				// Time out expected hanger is not arrived
				IF (me.SubStateMachine.udiTimeInState_ms > SIf.Par.udiTimeOutHRU_Hanger_ms) THEN	// Hanger Rotation Unit time out waiting
					pfbAlarmCtrl^.setAlarm(CIf.Info.intCtrlId,4,0,ADR(SIf.Alm),E_AlmState.RST,CIf.Job.eMe_ActivAlmClass);
					me.SubStateMachine.intStateNext := cSTA_SUB_ERROR;
				END_IF
		//--------------------------------------------------------------------------------------
			cSTA_SUB_WAIT_WITH_HANGER:
				IF (me.SubStateMachine.intState<>me.SubStateMachine.intStateLastCycle) THEN
					me.SubStateMachine.intStateLastCycle := me.SubStateMachine.intState;
				END_IF
				
				// State Change Condition
				// Check error if possible
				IF (me.SubStateMachine.udiTimeInState_ms >= SIf.Par.udiWaitForRotate_ms) THEN
					me.SubStateMachine.intStateNext := cSTA_SUB_ROTATE;
				END_IF
		//--------------------------------------------------------------------------------------
			cSTA_SUB_ROTATE:
				IF (me.SubStateMachine.intState<>me.SubStateMachine.intStateLastCycle) THEN
					me.SubStateMachine.intStateLastCycle := me.SubStateMachine.intState;
					SIf.Out.bolRotate.intern := NOT SIf.Out.bolRotate.intern;	// Rotate in other direction
				END_IF
				
				
				// State Change Condition
				// Check error if possible
				IF (me.SubStateMachine.udiTimeInState_ms >= SIf.Par.udiRotateTime_ms) THEN
					me.SubStateMachine.intStateNext := cSTA_SUB_EJECT;
				END_IF
		//--------------------------------------------------------------------------------------
			cSTA_SUB_EJECT:
				IF (me.SubStateMachine.intState<>me.SubStateMachine.intStateLastCycle) THEN
					me.SubStateMachine.intStateLastCycle := me.SubStateMachine.intState;
				END_IF
				
				SIf.Out.bolEject.intern := TRUE;	// Eject Cylinder Valve
				
				// Simulation
				IF (CIf.SwCfg.bolSimulation) THEN
					SIf.In.bolHangerDetected.intern := FALSE; // Hanger is leaving the HRU
				END_IF
				
				// State Change Condition
				// Check error if possible
				IF (me.SubStateMachine.udiTimeInState_ms > SIf.Par.udiEjectTime_ms) THEN
					IF (SIf.In.bolHangerDetected.intern) THEN
					// sensor Hanger detected always on
						pfbAlarmCtrl^.setAlarm(CIf.Info.intCtrlId,3,0,ADR(SIf.Alm),E_AlmState.RST,CIf.Job.eMe_ActivAlmClass);
						me.SubStateMachine.intStateNext := cSTA_SUB_ERROR;
					ELSE
						// Hanger ejected
						me.SubStateMachine.intStateNext := cSTA_SUB_RETRACT;
					END_IF
				END_IF
		//--------------------------------------------------------------------------------------
			cSTA_SUB_RETRACT:
				IF (me.SubStateMachine.intState<>me.SubStateMachine.intStateLastCycle) THEN
					me.SubStateMachine.intStateLastCycle := me.SubStateMachine.intState;
				END_IF
				
				SIf.Out.bolEject.intern := FALSE;	// Eject Cylinder Valve

				// State Change Condition
				// Check error if possible
				IF (me.SubStateMachine.udiTimeInState_ms >= SIf.Par.udiRetractTime_ms) THEN
					me.SubStateMachine.intStateNext := cSTA_SUB_DONE;
				END_IF
		//--------------------------------------------------------------------------------------
			cSTA_SUB_DONE:
				//CIf.Job.intACmd:=cSTA_DONE; 	// Not necessary
				;								// do nothing, just for state change
		//--------------------------------------------------------------------------------------
			cSTA_SUB_ERROR:
				IF (me.SubStateMachine.intState<>me.SubStateMachine.intStateLastCycle) THEN
					me.SubStateMachine.intStateLastCycle := me.SubStateMachine.intState;
				END_IF
				
				SIf.Out.bolEject.intern := FALSE;	// Eject Cylinder Valve
				
				// State Change Condition
				// No change, going over an other main state
		//--------------------------------------------------------------------------------------
		END_CASE
		
		// Do in every cycle
		CIf.Job.strSubState := THIS^.getCmdState(intCmdState:=me.SubStateMachine.intState,bolState:=TRUE);
		IF (me.SubStateMachine.intState<>me.SubStateMachine.intStateNext) THEN
			me.SubStateMachine.intState := me.SubStateMachine.intStateNext;  // set next state for next cycle
			me.SubStateMachine.udiTimeInState_ms := 0; // reset timer
			// log state change -> open point
		ELSE
			// increment time in state	
			me.SubStateMachine.udiTimeInState_ms := me.SubStateMachine.udiTimeInState_ms + me.FUBInfo.udiSample_ms;
		END_IF
		
				
		// State Change Condition	
		IF me.SubStateMachine.intState = cSTA_SUB_ERROR THEN
			me.StateMachine.intStateNext :=  cSTA_ERROR;
		ELSIF(me.SubStateMachine.intState = cSTA_SUB_DONE) THEN
			me.StateMachine.intStateNext := cSTA_RUN;
		ELSIF((me.SubStateMachine.intState = cSTA_SUB_WAIT_FOR_JOB) AND(me.intCmd=cCMD_STOP)) THEN
			me.StateMachine.intStateNext := cSTA_STOPBusy;
		//ELSIF((me.SubStateMachine.intState = cSTA_SUB_WAIT_FOR_JOB) AND(me.intCmd=cCMD_OFF)) THEN // Done by BaseCtrl.Always
		//	me.StateMachine.intStateNext := cSTA_OFFBusy;
		END_IF
	END_IF


//--------------------------------------------------------------------------------------
// Exit action
	IF (me.StateMachine.intState<>me.StateMachine.intStateNext) THEN
		;
	END_IF
END_METHOD

METHOD PROTECTED sta_STOP : BOOL
// state implemetation
//--------------------------------------------------------------------------------------
// Entry action
	IF (me.StateMachine.intState<>me.StateMachine.intStateLastCycle) THEN
		me.StateMachine.intStateLastCycle := me.StateMachine.intState;
		
	END_IF


//--------------------------------------------------------------------------------------
// Cyclic action
	IF (me.StateMachine.intState=me.StateMachine.intStateLastCycle) THEN
		
		;
		
		
		// State Change Condition
		IF (me.intCmd=cCMD_OFF) THEN
			// sensor retract always on cylinder
			me.StateMachine.intStateNext :=  cSTA_OFFBusy;
		ELSIF (me.intCmd=cCMD_EJECT) THEN 
			me.StateMachine.intStateNext := cSTA_EJECTBusy;
		ELSIF(me.intCmd=cCMD_RETRACT) THEN
			me.StateMachine.intStateNext := cSTA_RETRACTBusy;
		ELSIF(me.intCmd=cCMD_ROTATE) THEN
			me.StateMachine.intStateNext := cSTA_ROTATEBusy;
		ELSIF (me.intCmd=cCMD_RUN) THEN
			me.StateMachine.intStateNext := cSTA_RUNBusy;
		END_IF
	END_IF




//--------------------------------------------------------------------------------------
// Exit action
	IF (me.StateMachine.intState<>me.StateMachine.intStateNext) THEN
		;
	END_IF
END_METHOD

METHOD PROTECTED sta_STOPBusy : BOOL
// state implemetation
//--------------------------------------------------------------------------------------
// Entry action
	IF (me.StateMachine.intState<>me.StateMachine.intStateLastCycle) THEN
		me.StateMachine.intStateLastCycle := me.StateMachine.intState;
		
	END_IF


//--------------------------------------------------------------------------------------
// Cyclic action
	IF (me.StateMachine.intState=me.StateMachine.intStateLastCycle) THEN
		
		// switch off?
		// SIf.Out.bolEject.intern := FALSE;	// Eject Cylinder Valve
		
		// State Change Condition
		IF (FALSE) THEN
			;
		ELSIF (TRUE) THEN
			me.StateMachine.intStateNext := cSTA_STOP;
		END_IF
	END_IF




//--------------------------------------------------------------------------------------
// Exit action
	IF (me.StateMachine.intState<>me.StateMachine.intStateNext) THEN
		;
	END_IF
END_METHOD

METHOD PROTECTED StateMachine : BOOL
SUPER^.StateMachine();

// main statemachine of base controller
CASE me.StateMachine.intState OF
	cSTA_ROTATEBusy: 
        THIS^.sta_ROTATEBusy();
    cSTA_ROTATE: 
        THIS^.sta_ROTATE();
	cSTA_RETRACTBusy: 
        THIS^.sta_RETRACTBusy();
    cSTA_RETRACT: 
        THIS^.sta_RETRACT();
    cSTA_EJECTBusy:				// Eject 
        THIS^.sta_EJECTBusy();
    cSTA_EJECT: 
        THIS^.sta_EJECT();
	cSTA_RUNBusy: 
        THIS^.sta_RUNBusy();	// Auto (Wait - Rotate - Eject - Retract)
    cSTA_RUN: 
        THIS^.sta_RUN();
	cSTA_STOPBusy: 				// Rotate rests in his Position, Ejector in Retract Position
        THIS^.sta_STOPBusy();
    cSTA_STOP: 
        THIS^.sta_STOP();
		
END_CASE;
END_METHOD

END_FUNCTION_BLOCK

// POUs/Controller/Lvl0/JUN (Junction)/FB_JUN
FUNCTION_BLOCK FB_JUN EXTENDS FB_CtrlBase
VAR_INPUT
	In_bolPassed: BOOL;
END_VAR
VAR_OUTPUT
	Out_bolOpen: BOOL;
END_VAR
VAR
	/// Specific interface struct for public access
	SIf: T_Ctrl_SIf_JUN;
	/// Function specific variables
	bolfpRelease: BOOL;
	/// Job for checking the sensor
	bolCheckPass: BOOL;
	/// standard Loop variable
	uinI: UINT;
	/// Loop Variable for Hashtable
	intLoopHashtable: INT;
	/// Index to next job in Hashtable
	intNextHastableIdx: INT;
	/// Index to next job in Hashtable
	intActHastableIdx: INT;
	/// Calculated position to open junction
	dinNextOpenPosition_um: DINT;
	/// Calculated position to close junction
	dinNextClosePosition_um: DINT;
	///Last new position value from parent
	dinTransportPositionOld_um: DINT;
	///Position correction in faster Task cycletime
	dinPositionCorrection_um: DINT;
	///Position of the tag
	dinTagPosition_um: DINT;
	///Difference from actual Tag Position to junction
	dinPositionDifference_um: DINT;
	/// Rising edge of passed sensor
	bolFpPassed: BOOL;
	/// Array to check every hanger passed the sensor
	aCheckPassingTime: ARRAY[0..9] OF T_JUN_OutfeedCheck;
	/// Size of Array Check Passing
	intSizeCheckPassing: INT;
	/// Index for the check passing array
	intIndexCheckPassing: INT;
	/// Temporary Value
	udiValue: UDINT;
	/// Temporary Value
	uinValue: UINT;
END_VAR
VAR CONSTANT
	///sub States for RELEASE Function
	cSTA_SUB_INITIALIZED: INT := 500;
	cSTA_SUB_WAIT_FOR_JOB: INT := 501;
	cSTA_SUB_OPEN: INT := 502;
	cSTA_SUB_CLOSE: INT := 506;
	cSTA_SUB_ERROR: INT := 598;
	cSTA_SUB_FINISHED: INT := 600;
END_VAR

(*__________________________________________________________________________________________________
¦	
¦	Vistaprint Schweiz GmbH
¦	CH - 8401 Winterthur
¦
¦	www.vistaprint.ch - info@vistaprint.ch
¦___________________________________________________________________________________________________

Function desription:
Junction to release hanges out of the transport belt 


History:
Version		Date			Author		Comment
---------------------------------------------------------------------------------------------------
0.00.1		22.08.2013		AVME/PRE	Start history
0.00.2		19.09.2013		AVME/PRE	Implement new Base Concept
0.00.3		02.10.2013		VP/MK,RE	Fixed multiplication issues (cast INT to REAL before division)
0.00.4		10.12.2013		AVME/MRU	Reset aCheckPassing time at exit of sta_RUN
0.00.5		03.02.2014		AVME/MRU	Changed 'timeout passed sensor does not detect the hanger' to INFO

___________________________________________________________________________________________________*)


IF (me.bolActivate) THEN // cyclic call enabled
	IF (CIf.Info.bolInitDone=FALSE) THEN // first cycle -> init
		CtrlInit();
		CIf.Info.bolInitDone := TRUE;
	ELSE
		CycleStartDuty();
	
		Always();
		
		StateMachine();
		
		CycleEndDuty();
	END_IF
END_IF;

METHOD PROTECTED Always : BOOL
IF (me.bolChangeBackToAUTO=TRUE) THEN // switch mode to automatic switch off controller
	//me.StateMachine.intStateNext := cSTA_OFFBusy;
	me.bolChangeBackToAUTO := FALSE; // for cylinder no change to off when switch to automatic!!
END_IF

SUPER^.Always();

// ----------------------------------------------------------------------------------
// cyclic actions outside of statemachine
IF (me.StateMachine.intState<>cSTA_SINGLE_ANSWER) THEN
	SIf.Cur.bolPassed := SIf.In.bolPassed.intern;
	SIf.Cur.bolOpen := SIf.Out.bolOpen.intern;

	; // always error supervision
	
END_IF

// Always change actions in Base Library
// ----------------------------------------------------------------------------------
// overrule error always from base -> no EOFF State!! in EOFF go to OFF
IF (me.StateMachine.intStateNext = cSTA_EOFFBusy) THEN
	IF (me.StateMachine.intState=cSTA_OFF) THEN
		me.StateMachine.intStateNext := cSTA_OFF;
	ELSE // stay in OFF
		me.StateMachine.intStateNext := cSTA_OFFBusy;
	END_IF
END_IF
END_METHOD

METHOD FB_init : BOOL
VAR_INPUT
	///if TRUE, the retain variables are initialized (warm start / cold start)
	bInitRetains: BOOL;
	///if TRUE, the instance afterwards gets moved into the copy code (online change)
	bInCopyCode: BOOL;
END_VAR
VAR
	ii: UINT;
END_VAR
//------------------------------------------------------------------------------------------------------------------------
// to manually change in new FUB implementation!!!
// define valid commands for this controller
FOR ii:= 0 TO (SIZEOF(CIf.Job.aCmdList)/SIZEOF(CIf.Job.aCmdList[0])-1) BY 1 DO
	IF (CIf.Job.aCmdList[ii].intCmd=cCMD_INITIALIZED) THEN
		// found first empty array element
		EXIT;
	END_IF
END_FOR
CIf.Job.aCmdList[ii].intCmd := cCMD_STOP;
CIf.Job.aCmdList[ii].strName := 'Stop'; 
CIf.Job.aCmdList[ii].bolAvailable := TRUE;
ii := ii +1;
CIf.Job.aCmdList[ii].intCmd := JUN_CmdState.cCMD_RELEASE_ALL;
CIf.Job.aCmdList[ii].strName := 'Release All';
CIf.Job.aCmdList[ii].bolAvailable := TRUE;
ii := ii +1;
CIf.Job.aCmdList[ii].intCmd := JUN_CmdState.cCMD_RELEASE; // for test simulation single answer
CIf.Job.aCmdList[ii].strName := 'Release';
CIf.Job.aCmdList[ii].bolAvailable := TRUE;
ii := ii +1;
CIf.Job.aCmdList[ii].intCmd := cCMD_RUN;
CIf.Job.aCmdList[ii].strName := 'Run'; 
CIf.Job.aCmdList[ii].bolAvailable := TRUE;
ii := ii +1;
CIf.Job.aCmdList[ii].intCmd := cCMD_STOP;
CIf.Job.aCmdList[ii].strName := 'Stop'; 
CIf.Job.aCmdList[ii].bolAvailable := TRUE;
ii := ii +1;

// set name of class/typ
CIf.Info.strType := 'FB_JUN'; 

// set alarm class
SIf.Alm[1].eAlmClass := E_AlmClass.INFO;
SIf.Alm[1].strText := 'timeout passed sensor does not detect the hanger'; 
SIf.Alm[2].eAlmClass := E_AlmClass.INFO;
SIf.Alm[2].strText := 'RUN not possible, no Hashtable';
SIf.Alm[3].eAlmClass := E_AlmClass.INFO;
SIf.Alm[3].strText := 'Open not possible, destination is full';
SIf.Alm[4].eAlmClass := E_AlmClass.TSTOP;
SIf.Alm[4].strText := 'interlock open - movement stopped';


//*******************************************************************************
// initial values
//*******************************************************************************

// software configuration
CIf.SwCfg.bolExist := TRUE;
CIf.SwCfg.bolSimulation := FALSE;

// parmeter
SIf.Par.udiOpenTime_ms := 20;
SIf.Par.udiCloseTime_ms := 10;
SIf.Par.udiPassTime_ms := 6000;

SIf.Par.udiSimPassTime_ms := SIf.Par.udiPassTime_ms/2;

SIf.Par.dinPosition_um := 10000000;
SIf.Par.dinOpenWay_um := 200000;

//*******************************************************************************
// initial values childes
//*******************************************************************************
END_METHOD

METHOD PROTECTED getCmdState : STRING
VAR_INPUT
	intCmdState: INT;
	bolState: BOOL;
END_VAR
getCmdState := SUPER^.getCmdState(intCmdState:=intCmdState,bolState:=bolState); // get global/base defined cmds/states
IF (getCmdState='') THEN // global not defined get local
	// get string cmd/state string information in runtime
	IF (bolState=FALSE) THEN
		// cmd's
		CASE intCmdState OF
			JUN_CmdState.cCMD_RELEASE_ALL: 
				getCmdState := 'cCMD_RELEASE_ALL';
			JUN_CmdState.cCMD_RELEASE: 
				getCmdState := 'cCMD_RELEASE';
		END_CASE;
	ELSE
	
	// cmd's
		CASE intCmdState OF
			cSTA_RUNBusy: 
				THIS^.sta_RUNBusy();
			cSTA_RUN: 
				THIS^.sta_RUN();
			cSTA_STOPBusy: 
				THIS^.sta_STOPBusy();
			cSTA_STOP: 
				THIS^.sta_STOP();
			JUN_CmdState.cSTA_RELEASE_ALLBusy: 
				THIS^.sta_RELEASE_ALLBusy();
			JUN_CmdState.cSTA_RELEASE_ALL: 
				THIS^.sta_RELEASE_ALL();
			JUN_CmdState.cSTA_RELEASEBusy: 
				THIS^.sta_RELEASEBusy();
			JUN_CmdState.cSTA_RELEASE: 
				THIS^.sta_RELEASE();
				
			// SUB States
			cSTA_SUB_INITIALIZED:
				getCmdState := 'cSTA_SUB_INITIALIZED';
			cSTA_SUB_WAIT_FOR_JOB:
				getCmdState := 'cSTA_SUB_WAIT_FOR_JOB';
			cSTA_SUB_OPEN:
				getCmdState := 'cSTA_SUB_OPEN';
			cSTA_SUB_CLOSE:
				getCmdState := 'cSTA_SUB_CLOSE';
			cSTA_SUB_ERROR:
				getCmdState := 'cSTA_SUB_ERROR';
			cSTA_SUB_FINISHED:
				getCmdState := 'cSTA_SUB_FINISHED';
		END_CASE;
	END_IF
END_IF
END_METHOD

METHOD getCtrlSIf : POINTER TO T_Ctrl_SIf_JUN
getCtrlSIf := ADR(SIf);
END_METHOD

METHOD PROTECTED IoInBridge : BOOL
// digitale and analoge inputs read from hardware or forcing

SIf.In.bolPassed.map := THIS^.In_bolPassed;

IF (CIf.SwCfg.bolSimulation = FALSE) THEN
	getInBol(CIf.Job.bolIoForce,ADR(SIf.In.bolPassed));
	//ctrl.In.bol_PosSwitchBasicDefTyp.intern := getInBol(ctrl.ifc.Job.bol_Force ,ADR(ctrl.In.bol_PosSwitchBasicDefTyp);
ELSE
	//simulation of global IO
END_IF
END_METHOD

METHOD PROTECTED IoOutBridge : BOOL
// digitale and analoge inputs read from hardware or forcing
IF (CIf.SwCfg.bolSimulation = FALSE) THEN
	setOutBol(CIf.Job.bolIoForce ,ADR(SIf.Out.bolOpen));
	
	// check interlocks to prevent damages
	IF (CIf.Job.bolIlkOverwrite=FALSE) THEN
		IF (SIf.Ilk.bolOpen=TRUE) THEN
			// switch off?
			IF (SIf.Out.bolOpen.map = TRUE) THEN
				// Set alarm: SIf.Alm[4].strText := 'interlock open - movement stopped';
				pfbAlarmCtrl^.setAlarm(CIf.Info.intCtrlId,4,0,ADR(SIf.Alm),E_AlmState.RST,CIf.Job.eMe_ActivAlmClass);
			END_IF
			SIf.Out.bolOpen.map := FALSE;
		END_IF	
	END_IF
	THIS^.Out_bolOpen := SIf.Out.bolOpen.map;
END_IF
END_METHOD

METHOD PROTECTED sta_ERROR : BOOL
// state implemetation
//--------------------------------------------------------------------------------------
// Entry action
	IF (me.StateMachine.intState<>me.StateMachine.intStateLastCycle) THEN
		me.StateMachine.intStateHistory := me.StateMachine.intStateLastCycle; // -> possibillity to go back to state before error
		me.StateMachine.intStateLastCycle := me.StateMachine.intState;
		
	END_IF


//--------------------------------------------------------------------------------------
// Cyclic action
	IF (me.StateMachine.intState=me.StateMachine.intStateLastCycle) THEN
		
		SIf.Out.bolOpen.intern := 0;
		
		
		// State Change Condition
		IF (CIf.Job.bolAlmReset = TRUE) THEN
			me.StateMachine.intStateNext := cSTA_ERRORQuit;
		END_IF
	END_IF




//--------------------------------------------------------------------------------------
// Exit action
	IF (me.StateMachine.intState<>me.StateMachine.intStateNext) THEN
		;
	END_IF
END_METHOD

METHOD PROTECTED sta_ERRORQuit : BOOL
// state implemetation
//--------------------------------------------------------------------------------------
// Entry action
	IF (me.StateMachine.intState<>me.StateMachine.intStateLastCycle) THEN
		me.StateMachine.intStateLastCycle := me.StateMachine.intState;
			FOR uinI := 0 TO (SIZEOF(aCheckPassingTime)/(SIZEOF(aCheckPassingTime[0]))-1) DO
				aCheckPassingTime[uinI].udiTime_ms := 0;
				aCheckPassingTime[uinI].intHTIndex := 0;
			END_FOR
	END_IF


//--------------------------------------------------------------------------------------
// Cyclic action
	IF (me.StateMachine.intState=me.StateMachine.intStateLastCycle) THEN
		
		;
		// evtl. wait time if reset of device is necessary and then decide to go to states or ERROR state
		IF (CIf.Job.bolAlmReset = TRUE) THEN
			CIf.Job.eMe_ActivAlmClass := E_AlmClass.NONE; // reset feedback channel for parent
			CIf.Job.bolAlmReset := FALSE;
		END_IF
		
		// State Change Condition
		IF (CIf.Job.bolAlmReset = FALSE) THEN
			IF (me.StateMachine.intStateHistory<=cSTA_PON) THEN
				me.StateMachine.intStateNext := cSTA_PONBusy;
			ELSIF(me.intCmd=cCMD_OFF) THEN
				me.StateMachine.intStateNext := cSTA_OFFBusy;
			ELSIF(me.intCmd=cCMD_RUN) OR (me.StateMachine.intStateHistory=cSTA_RUN) THEN
				me.StateMachine.intStateNext := cSTA_RUNBusy;
			ELSIF(me.intCmd=cCMD_STOP) THEN
				me.StateMachine.intStateNext := cSTA_STOPBusy;
			ELSIF(me.intCmd=JUN_CmdState.cCMD_RELEASE_ALL) THEN
				me.StateMachine.intStateNext := JUN_CmdState.cSTA_RELEASE_ALLBusy;
			ELSIF(me.intCmd=JUN_CmdState.cCMD_RELEASE) THEN
				me.StateMachine.intStateNext := JUN_CmdState.cSTA_RELEASEBusy;
			END_IF
		END_IF
	END_IF




//--------------------------------------------------------------------------------------
// Exit action
	IF (me.StateMachine.intState<>me.StateMachine.intStateNext) THEN
		;
	END_IF
END_METHOD

METHOD PROTECTED sta_OFF : BOOL
// state implemetation
//--------------------------------------------------------------------------------------
// Entry action
	IF (me.StateMachine.intState<>me.StateMachine.intStateLastCycle) THEN
		me.StateMachine.intStateLastCycle := me.StateMachine.intState;
		
	END_IF


//--------------------------------------------------------------------------------------
// Cyclic action
	IF (me.StateMachine.intState=me.StateMachine.intStateLastCycle) THEN
		
		;
		
		
		// State Change Condition
		IF (me.Alarm.eActivAlmClass<>E_AlmClass.EOFF) AND (me.Alarm.eActivAlmClass<>E_AlmClass.OFF) THEN
			IF (me.intCmd=cCMD_STOP) THEN
				// sensor retract always on cylinder
				me.StateMachine.intStateNext :=  cSTA_STOPBusy;
			ELSIF (me.intCmd=JUN_CmdState.cCMD_RELEASE) THEN 
				me.StateMachine.intStateNext := JUN_CmdState.cSTA_RELEASEBusy;
			ELSIF(me.intCmd=JUN_CmdState.cCMD_RELEASE_ALL) THEN
				me.StateMachine.intStateNext := JUN_CmdState.cSTA_RELEASE_ALLBusy;
			ELSIF(me.intCmd=cCMD_RUN) THEN
				me.StateMachine.intStateNext := cSTA_RUNBusy;
			END_IF
		END_IF
	END_IF




//--------------------------------------------------------------------------------------
// Exit action
	IF (me.StateMachine.intState<>me.StateMachine.intStateNext) THEN
		;
	END_IF
END_METHOD

METHOD PROTECTED sta_OFFBusy : BOOL
// state implemetation
//--------------------------------------------------------------------------------------
// Entry action
	IF (me.StateMachine.intState<>me.StateMachine.intStateLastCycle) THEN
		me.StateMachine.intStateLastCycle := me.StateMachine.intState;
		
	END_IF


//--------------------------------------------------------------------------------------
// Cyclic action
	IF (me.StateMachine.intState=me.StateMachine.intStateLastCycle) THEN
		
		// switch VALVE off
		SIf.Out.bolOpen.intern := FALSE;
		
		
		
		// State Change Condition
		IF (FALSE) THEN
			;
		ELSIF (TRUE) THEN
			me.StateMachine.intStateNext := cSTA_OFF;
		END_IF
	END_IF




//--------------------------------------------------------------------------------------
// Exit action
	IF (me.StateMachine.intState<>me.StateMachine.intStateNext) THEN
		;
	END_IF
END_METHOD

METHOD PROTECTED sta_PON : BOOL
// state implemetation
//--------------------------------------------------------------------------------------
// Entry action
	IF (me.StateMachine.intState<>me.StateMachine.intStateLastCycle) THEN
		me.StateMachine.intStateLastCycle := me.StateMachine.intState;
		
	END_IF


//--------------------------------------------------------------------------------------
// Cyclic action
	IF (me.StateMachine.intState=me.StateMachine.intStateLastCycle) THEN
		
		;
		
		
		// State Change Condition
		IF(me.intCmd=cCMD_OFF) THEN
			me.StateMachine.intStateNext := cSTA_OFFBusy;
		ELSIF(me.intCmd=cCMD_RUN) THEN
			me.StateMachine.intStateNext := cSTA_OFFBusy;
		ELSIF(me.intCmd=cCMD_STOP) THEN
			me.StateMachine.intStateNext := cSTA_STOPBusy;
		ELSIF(me.intCmd=JUN_CmdState.cCMD_RELEASE) THEN
			me.StateMachine.intStateNext := JUN_CmdState.cSTA_RELEASEBusy;
		ELSIF (me.intCmd=JUN_CmdState.cCMD_RELEASE_ALL) THEN
			me.StateMachine.intStateNext := JUN_CmdState.cSTA_RELEASE_ALLBusy;
		END_IF
	END_IF




//--------------------------------------------------------------------------------------
// Exit action
	IF (me.StateMachine.intState<>me.StateMachine.intStateNext) THEN
		;
	END_IF
END_METHOD

METHOD PROTECTED sta_RELEASE : BOOL
// state implemetation
//--------------------------------------------------------------------------------------
// Entry action
	IF (me.StateMachine.intState<>me.StateMachine.intStateLastCycle) THEN
		me.StateMachine.intStateLastCycle := me.StateMachine.intState;
		
	END_IF


//--------------------------------------------------------------------------------------
// Cyclic action
	IF (me.StateMachine.intState=me.StateMachine.intStateLastCycle) THEN
		// Check the CMD change for next release
		IF (me.intCmd<>JUN_CmdState.cCMD_RELEASE) THEN
			bolfpRelease := FALSE;		// Only start once the release if cmd is still the same
		END_IF
	
	
		// Simulation
		
		// State Change Condition
		IF(me.intCmd=cCMD_STOP) THEN
			me.StateMachine.intStateNext := cSTA_STOPBusy;
		ELSIF(me.intCmd=JUN_CmdState.cCMD_RELEASE_ALL) THEN
			me.StateMachine.intStateNext := JUN_CmdState.cSTA_RELEASE_ALLBusy;
		ELSIF((me.intCmd=JUN_CmdState.cCMD_RELEASE) AND (bolfpRelease = FALSE)) THEN
			me.StateMachine.intStateNext := JUN_CmdState.cSTA_RELEASEBusy;			
		ELSIF(me.intCmd=cCMD_RUN) THEN
			me.StateMachine.intStateNext := cSTA_STOPBusy;			
		END_IF
	END_IF




//--------------------------------------------------------------------------------------
// Exit action
	IF (me.StateMachine.intState<>me.StateMachine.intStateNext) THEN
		bolfpRelease := FALSE;		// Only start once the release if cmd is still the same
	END_IF
END_METHOD

METHOD PROTECTED sta_RELEASE_ALL : BOOL
// state implemetation
//--------------------------------------------------------------------------------------
// Entry action
	IF (me.StateMachine.intState<>me.StateMachine.intStateLastCycle) THEN
		me.StateMachine.intStateLastCycle := me.StateMachine.intState;
		
		fbSimulationTimer.IN := FALSE;
		fbSimulationTimer.PT := UDINT_TO_TIME(SIf.Par.udiSimPassTime_ms);
		fbSimulationTimer(); // set time/reset timer
		fbSimulationTimer.IN := TRUE; // start timer

	END_IF


//--------------------------------------------------------------------------------------
// Cyclic action
	IF (me.StateMachine.intState=me.StateMachine.intStateLastCycle) THEN

		// Simulation
		IF (CIf.SwCfg.bolSimulation) THEN
			fbSimulationTimer(); // simulation time
			IF (fbSimulationTimer.Q) THEN
				fbSimulationTimer.IN := FALSE;
				IF SIf.In.bolPassed.intern = FALSE THEN
					SIf.In.bolPassed.intern := TRUE;
				ELSE
					SIf.In.bolPassed.intern := FALSE;
				END_IF
			ELSE
				fbSimulationTimer.IN := TRUE; // start timer
			END_IF
		END_IF

		
		// State Change Condition
		IF(me.intCmd=cCMD_STOP) THEN
			me.StateMachine.intStateNext := cSTA_STOPBusy;
		ELSIF(me.intCmd=JUN_CmdState.cCMD_RELEASE) THEN
			me.StateMachine.intStateNext := JUN_CmdState.cSTA_RELEASEBusy;
		ELSIF(me.intCmd=cCMD_RUN) THEN
			me.StateMachine.intStateNext := cSTA_STOPBusy;
		END_IF
	END_IF




//--------------------------------------------------------------------------------------
// Exit action
	IF (me.StateMachine.intState<>me.StateMachine.intStateNext) THEN
		;
	END_IF
END_METHOD

METHOD PROTECTED sta_RELEASE_ALLBusy : BOOL
// state implemetation
//--------------------------------------------------------------------------------------
// Entry action
	IF (me.StateMachine.intState<>me.StateMachine.intStateLastCycle) THEN
		me.StateMachine.intStateLastCycle := me.StateMachine.intState;
		
		SIf.Out.bolOpen.intern := TRUE;
	END_IF


//--------------------------------------------------------------------------------------
// Cyclic action
	IF (me.StateMachine.intState=me.StateMachine.intStateLastCycle) THEN

		// Simulation

		
		// State Change Condition
		IF (me.StateMachine.udiTimeInState_ms > SIf.Par.udiOpenTime_ms) THEN
			me.StateMachine.intStateNext := JUN_CmdState.cSTA_RELEASE_ALL;
		ELSIF(me.intCmd=cCMD_STOP) THEN
			me.StateMachine.intStateNext := cSTA_STOPBusy;
		ELSIF(me.intCmd=JUN_CmdState.cCMD_RELEASE) THEN
			me.StateMachine.intStateNext := JUN_CmdState.cSTA_RELEASEBusy;
		ELSIF(me.intCmd=cCMD_RUN) THEN
			me.StateMachine.intStateNext := cSTA_STOPBusy;
		END_IF
	END_IF




//--------------------------------------------------------------------------------------
// Exit action
	IF (me.StateMachine.intState<>me.StateMachine.intStateNext) THEN
		;
	END_IF
END_METHOD

METHOD PROTECTED sta_RELEASEBusy : BOOL
// state implemetation
//--------------------------------------------------------------------------------------
// Entry action
	IF (me.StateMachine.intState<>me.StateMachine.intStateLastCycle) THEN
		me.StateMachine.intStateLastCycle := me.StateMachine.intState;
					
		me.SubStateMachine.intState := cSTA_SUB_INITIALIZED; // init sub state machine
		me.SubStateMachine.intStateNext := cSTA_SUB_INITIALIZED; // init sub state machine
		bolfpRelease := TRUE;		// Only start once the release if cmd is still the same
	END_IF


//--------------------------------------------------------------------------------------
// Cyclic action
	IF (me.StateMachine.intState=me.StateMachine.intStateLastCycle) THEN
	

		//--------------------------------------------------------------------------------------
		// sub state machine for sequence
		CASE me.SubStateMachine.intState OF
			//--------------------------------------------------------------------------------------
			cSTA_SUB_INITIALIZED:
					// State Change Condition
					// Simulation
					IF (CIf.SwCfg.bolSimulation) THEN
							SIf.In.bolPassed.intern := FALSE;
					END_IF

					// only release one tray if no jam is at the stopper
					IF (SIf.In.bolPassed.intern = FALSE) THEN
						me.SubStateMachine.intStateNext := cSTA_SUB_OPEN;
						// Start Timer
						fbSimulationTimer.IN := FALSE;
						fbSimulationTimer.PT := UDINT_TO_TIME(SIf.Par.udiSimPassTime_ms);
						fbSimulationTimer(); // set time/reset timer
						fbSimulationTimer.IN := TRUE; // start timer
	
					ELSE
						// SIf.Alm[3].strText := 'Open not possible, destination is full';
						pfbAlarmCtrl^.setAlarm(CIf.Info.intCtrlId,3,0,ADR(SIf.Alm),E_AlmState.RST,CIf.Job.eMe_ActivAlmClass);	
					END_IF
					
			//--------------------------------------------------------------------------------------
			cSTA_SUB_OPEN:
					SIf.Out.bolOpen.intern := TRUE;
					
					// Simulation
					IF (CIf.SwCfg.bolSimulation) THEN
						fbSimulationTimer(); // simulation time
						IF (fbSimulationTimer.Q) THEN
							SIf.In.bolPassed.intern := TRUE;						
						END_IF
					END_IF
					
					
				// State Change Condition
					// Check error if tray never reach the output
					IF (me.SubStateMachine.udiTimeInState_ms>SIf.Par.udiPassTime_ms) THEN
						// Set Alarm: SIf.Alm[1].strText := 'timeout passed sensor does not detect the hanger'; 
						pfbAlarmCtrl^.setAlarm(CIf.Info.intCtrlId,1,0,ADR(SIf.Alm),E_AlmState.RST,CIf.Job.eMe_ActivAlmClass);
						me.SubStateMachine.intStateNext := cSTA_ERROR;
					// Check if tray allready passed
					ELSIF (SIf.In.bolPassed.intern = TRUE) THEN
						me.SubStateMachine.intStateNext := cSTA_SUB_CLOSE;
					END_IF

					
			//--------------------------------------------------------------------------------------
			cSTA_SUB_CLOSE:
					SIf.Out.bolOpen.intern := FALSE;
					
					// Simulation
					
					
					// State Change Condition
					// Check error if retracted position not reached
					IF (me.SubStateMachine.udiTimeInState_ms > SIf.Par.udiCloseTime_ms) THEN
						me.SubStateMachine.intStateNext := cSTA_SUB_FINISHED;
						// Simulation
						IF (CIf.SwCfg.bolSimulation) THEN
								SIf.In.bolPassed.intern := FALSE;
						END_IF
					END_IF
				
			//--------------------------------------------------------------------------------------
			cSTA_SUB_ERROR:
					SIf.Out.bolOpen.intern := FALSE;
					
					// State Change Condition
					// No change, going over an other main state
					
			//--------------------------------------------------------------------------------------
			cSTA_SUB_FINISHED:
					;
					
		END_CASE
		
		// State Change Condition
		// Check error if retracted position not reached
		IF me.SubStateMachine.intState = cSTA_SUB_ERROR THEN
			me.StateMachine.intStateNext :=  cSTA_ERROR;
		ELSIF (me.SubStateMachine.intState = cSTA_SUB_FINISHED) THEN
			me.StateMachine.intStateNext := JUN_CmdState.cSTA_RELEASE;
		ELSIF(me.intCmd=cCMD_STOP) THEN
			me.StateMachine.intStateNext := cSTA_STOPBusy;
		ELSIF(me.intCmd=JUN_CmdState.cCMD_RELEASE_ALL) THEN
			me.StateMachine.intStateNext := JUN_CmdState.cSTA_RELEASE_ALLBusy;
		ELSIF(me.intCmd=cCMD_RUN) THEN
			me.StateMachine.intStateNext := cSTA_STOPBusy;			
		END_IF
	END_IF




//--------------------------------------------------------------------------------------
// Exit action
	IF (me.StateMachine.intState<>me.StateMachine.intStateNext) THEN
		;
	END_IF
END_METHOD

METHOD PROTECTED sta_RUN : BOOL
// state implemetation
//--------------------------------------------------------------------------------------
// Entry action
	IF (me.StateMachine.intState<>me.StateMachine.intStateLastCycle) THEN
		me.StateMachine.intStateLastCycle := me.StateMachine.intState;
			
		me.SubStateMachine.intState := cSTA_SUB_WAIT_FOR_JOB; // init sub state machine
		me.SubStateMachine.intStateNext := cSTA_SUB_WAIT_FOR_JOB; // init sub state machine
		bolfpRelease := TRUE;		// Only start once the release if cmd is still the same
		fbSimulationTimer.PT := UDINT_TO_TIME(SIf.Par.udiSimPassTime_ms);
		fbSimulationTimer(); // set time/reset timer

	END_IF


//--------------------------------------------------------------------------------------
// Cyclic action
	IF (me.StateMachine.intState=me.StateMachine.intStateLastCycle) THEN
		// Simulation
		IF (CIf.SwCfg.bolSimulation) THEN
			fbSimulationTimer(); // set time/reset timer
			IF SIf.Out.bolOpen.intern = TRUE THEN 
				fbSimulationTimer.IN := TRUE;
			ELSIF (SIf.Out.bolOpen.intern = FALSE) AND (fbSimulationTimer.Q = TRUE) THEN
				fbSimulationTimer.IN := FALSE;				
			END_IF
			IF fbSimulationTimer.Q = TRUE THEN
				SIf.In.bolPassed.intern := TRUE;
			ELSE
				SIf.In.bolPassed.intern := FALSE;
			END_IF
		END_IF
		
		//--------------------------------------------------------------------------------------
		// Always RUN actions
		
		// If this task is in faster cycle then the parent, calculate internal position more exactly during the taskcycle
		IF dinTransportPositionOld_um <> SIf.Cur.dinTransportPosition_um THEN
			SIf.Cur.dinTransportPositionCalc_um := SIf.Cur.dinTransportPosition_um;
			dinTransportPositionOld_um := SIf.Cur.dinTransportPosition_um;
			dinPositionCorrection_um := 0;
		ELSE
			dinPositionCorrection_um := dinPositionCorrection_um + LREAL_TO_DINT(DINT_TO_LREAL(SIf.Cur.dinTransportspeed_um_s) * UDINT_TO_LREAL(me.FUBInfo.udiSample_ms) / 1000.0 );
			SIf.Cur.dinTransportPositionCalc_um := dinTransportPositionOld_um + dinPositionCorrection_um;
		END_IF
		
		// Check hashtable if there is a job
		dinPositionDifference_um := SIf.Par.dinPosition_um; // Set maximal value to search the smalles one
		// Loop through the hashtable
		FOR intLoopHashtable := 0 TO cintMaxDecisions DO
			// Check if the hashtable entry is for this target
			IF SIf.par.pTblDecision^[intLoopHashtable].stDecision.dinTarget = SIf.Cfg.dinTargetNr THEN
				// Check if this job is on the way to the junction
				IF SIf.par.pTblDecision^[intLoopHashtable].eState = E_DecisionState.WayToJunction THEN
					// Check if Tag is not already driven too much
					IF SIf.par.pTblDecision^[intLoopHashtable].dinActPos_um > (SIf.Par.dinPosition_um + SIf.Par.dinOpenWay_um) THEN
						// If driven to much, wait for next passing
						SIf.par.pTblDecision^[intLoopHashtable].eState := E_DecisionState.Wait;
					ELSE
						// Check if it is the nearest tag
						IF 	dinPositionDifference_um > SIf.Par.dinPosition_um - SIf.par.pTblDecision^[intLoopHashtable].dinActPos_um THEN
							dinPositionDifference_um := SIf.Par.dinPosition_um - SIf.par.pTblDecision^[intLoopHashtable].dinActPos_um;
							intNextHastableIdx := intLoopHashtable;
						END_IF
					END_IF
				END_IF
			END_IF
		END_FOR
		
		// Calculate the exactly position of the next Tag to Work with
		IF SIf.par.pTblDecision^[intNextHastableIdx].stDecision.dinTarget = SIf.Cfg.dinTargetNr 
			AND SIf.par.pTblDecision^[intNextHastableIdx].eState = E_DecisionState.WayToJunction THEN
			// Only calculate next position if a new job for this junction is ready
			dinPositionDifference_um := SIf.Par.dinPosition_um - SIf.par.pTblDecision^[intNextHastableIdx].dinActPos_um - dinPositionCorrection_um;
		ELSE	
			dinPositionDifference_um := SIf.Par.dinPosition_um;
		END_IF
		
		// Check the sensor for Timeout Error 
		// Array for more than one hanger check, if a hanger pass the junction, the value is set to 1
		// Every Value in the array > 0 would be cyclicle increased
		// If a value is higher than the maximum time, error occures
		// A rising edge of the sensor would cleare the oldest value
		
		// Delete old values
		IF ((SIf.In.bolPassed.intern = TRUE) AND (bolFpPassed = FALSE)) THEN
			bolFpPassed := TRUE;
			// Delete Check time from sensor from oldest value
			udiValue := 0;
			FOR uinI := 0 TO (SIZEOF(aCheckPassingTime)/(SIZEOF(aCheckPassingTime[0]))-1) DO
				IF aCheckPassingTime[uinI].udiTime_ms > udiValue THEN
					udiValue := aCheckPassingTime[uinI].udiTime_ms;
					uinValue := uinI;
				END_IF
			END_FOR
			// Reset oldest Value
			aCheckPassingTime[uinValue].udiTime_ms := 0;
			// Change state in hashtable from this value
			SIf.par.pTblDecision^[aCheckPassingTime[uinValue].intHTIndex].eState := E_DecisionState.DriveOut;
			SIf.par.pTblDecision^[aCheckPassingTime[uinValue].intHTIndex].dinActPos_um := -2;
			// Reset Index
			aCheckPassingTime[uinValue].intHTIndex := 0;		
			
		ELSIF (SIf.In.bolPassed.intern = FALSE) THEN
			bolFpPassed := FALSE;
		END_IF
		
		// Check every value
		FOR uinI := 0 TO (SIZEOF(aCheckPassingTime)/(SIZEOF(aCheckPassingTime[0]))-1) DO
			IF aCheckPassingTime[uinI].udiTime_ms > SIf.Par.udiPassTime_ms THEN
				// Set Alarm: SIf.Alm[1].strText := 'timeout passed sensor does not detect the hanger';
				pfbAlarmCtrl^.setAlarm(CIf.Info.intCtrlId,1,0,ADR(SIf.Alm),E_AlmState.RST,CIf.Job.eMe_ActivAlmClass);	
			ELSIF aCheckPassingTime[uinI].udiTime_ms > 0 THEN
				aCheckPassingTime[uinI].udiTime_ms := aCheckPassingTime[uinI].udiTime_ms + me.FUBInfo.udiSample_ms;
			END_IF
		END_FOR
			
		
		//--------------------------------------------------------------------------------------
		// sub state machine for sequence
		CASE me.SubStateMachine.intState OF
			//--------------------------------------------------------------------------------------
			cSTA_SUB_WAIT_FOR_JOB:
				IF (me.SubStateMachine.intState<>me.SubStateMachine.intStateLastCycle) THEN
					me.SubStateMachine.intStateLastCycle := me.SubStateMachine.intState;
				END_IF
				// State Change Condition
				// Simulation
				IF (CIf.SwCfg.bolSimulation) THEN
						SIf.In.bolPassed.intern := FALSE;
				END_IF
				
				// If reaction way (time*speed) is bigger then the rest of the way to the junction, open
				IF dinPositionDifference_um <= LREAL_TO_DINT( UDINT_TO_LREAL(SIf.Par.udiOpenTime_ms) * DINT_TO_LREAL(SIf.Cur.dinTransportspeed_um_s) ) / 1000.0 THEN
					// only release one tray if no jam is at the stopper
					IF (SIf.In.bolPassed.intern = FALSE) THEN
						// Save actual index
						me.SubStateMachine.intStateNext := cSTA_SUB_OPEN;
					ELSE
						// SIf.Alm[3].strText := 'Open not possible, destination is full';
						pfbAlarmCtrl^.setAlarm(CIf.Info.intCtrlId,3,0,ADR(SIf.Alm),E_AlmState.RST,CIf.Job.eMe_ActivAlmClass);	
					END_IF
				END_IF	
			//--------------------------------------------------------------------------------------
			cSTA_SUB_OPEN:
				IF (me.SubStateMachine.intState<>me.SubStateMachine.intStateLastCycle) THEN
					me.SubStateMachine.intStateLastCycle := me.SubStateMachine.intState;

					intActHastableIdx := intNextHastableIdx;
					SIf.par.pTblDecision^[intNextHastableIdx].eState := E_DecisionState.OnJunction;
					
					// Start the Sensor timeout check with write 1 into the checking Array to inrease the time
					IF aCheckPassingTime[intIndexCheckPassing].udiTime_ms = 0 THEN
						aCheckPassingTime[intIndexCheckPassing].udiTime_ms := 1;
						aCheckPassingTime[intIndexCheckPassing].intHTIndex := intActHastableIdx;
					END_IF
					
					// Increment the checking position 
					IF intIndexCheckPassing >= (SIZEOF(aCheckPassingTime)/SIZEOF(aCheckPassingTime[0]) - 1) THEN
						intIndexCheckPassing := 0;
					ELSE
						intIndexCheckPassing := intIndexCheckPassing + 1;
					END_IF

				END_IF
					
				SIf.Out.bolOpen.intern := TRUE;
					
				// Simulation
				IF (CIf.SwCfg.bolSimulation) THEN
					;
				END_IF
					
				// Check position
				IF (SIf.Par.dinPosition_um + SIf.Par.dinOpenWay_um <= SIf.par.pTblDecision^[intActHastableIdx].dinActPos_um + dinPositionCorrection_um) THEN
					IF SIf.par.pTblDecision^[intActHastableIdx].eState < E_DecisionState.Processed THEN
						// Only set to processe if not allready driven out
						SIf.par.pTblDecision^[intActHastableIdx].eState := E_DecisionState.Processed;
					END_IF					
					SIf.par.pTblDecision^[intActHastableIdx].dinActPos_um := -2;
				END_IF
					
				// State Change Condition
				// Check error if tray never reach the output
				IF (me.SubStateMachine.udiTimeInState_ms > SIf.Par.udiPassTime_ms) THEN
					// Set Alarm: SIf.Alm[1].strText := 'timeout passed sensor does not detect the hanger'; 
					pfbAlarmCtrl^.setAlarm(CIf.Info.intCtrlId,1,0,ADR(SIf.Alm),E_AlmState.RST,CIf.Job.eMe_ActivAlmClass);
					me.SubStateMachine.intStateNext := cSTA_ERROR;
				// Check if tray allready passed
				ELSIF (SIf.par.pTblDecision^[intActHastableIdx].eState > E_DecisionState.OnJunction) AND (dinPositionDifference_um < LREAL_TO_DINT ( UDINT_TO_LREAL(SIf.Par.udiOpenTime_ms) * DINT_TO_LREAL(SIf.Cur.dinTransportspeed_um_s) / 1000.0 ) ) THEN
					me.SubStateMachine.intStateNext := cSTA_SUB_OPEN;
				ELSIF (SIf.par.pTblDecision^[intActHastableIdx].eState > E_DecisionState.OnJunction) THEN	
					me.SubStateMachine.intStateNext := cSTA_SUB_CLOSE;
				END_IF

					
			//--------------------------------------------------------------------------------------
			cSTA_SUB_CLOSE:
				IF (me.SubStateMachine.intState<>me.SubStateMachine.intStateLastCycle) THEN
					me.SubStateMachine.intStateLastCycle := me.SubStateMachine.intState;
				END_IF
				
				SIf.Out.bolOpen.intern := FALSE;
					
				// Simulation
					
					
				// State Change Condition
				// Check error if retracted position not reached
				IF (TRUE) THEN
					me.SubStateMachine.intStateNext := cSTA_SUB_WAIT_FOR_JOB;
					// Simulation
					IF (CIf.SwCfg.bolSimulation) THEN
							SIf.In.bolPassed.intern := FALSE;
					END_IF
				END_IF
				
			//--------------------------------------------------------------------------------------
			cSTA_SUB_ERROR:
				IF (me.SubStateMachine.intState<>me.SubStateMachine.intStateLastCycle) THEN
					me.SubStateMachine.intStateLastCycle := me.SubStateMachine.intState;
				END_IF
				
				SIf.Out.bolOpen.intern := FALSE;
				
				// State Change Condition
				// No change, going over an other main state
					
		END_CASE
		
		
		// State Change Condition
		// Check error if retracted position not reached
		IF me.SubStateMachine.intState = cSTA_SUB_ERROR THEN
			me.StateMachine.intStateNext :=  cSTA_ERROR;
		ELSIF(me.intCmd=cCMD_STOP) THEN
			me.StateMachine.intStateNext := cSTA_STOPBusy;
		ELSIF(me.intCmd=JUN_CmdState.cCMD_RELEASE_ALL) THEN
			me.StateMachine.intStateNext := JUN_CmdState.cSTA_RELEASE_ALLBusy;		
		END_IF
	END_IF




//--------------------------------------------------------------------------------------
// Exit action
	IF (me.StateMachine.intState<>me.StateMachine.intStateNext) THEN
		// Reset aCheckPassingTime
		FOR uinI := 0 TO (SIZEOF(aCheckPassingTime)/(SIZEOF(aCheckPassingTime[0]))-1) DO
			aCheckPassingTime[uinI].udiTime_ms := 0;
			aCheckPassingTime[uinI].intHTIndex := 0;
		END_FOR;
	END_IF
END_METHOD

METHOD PROTECTED sta_RUNBusy : BOOL
// state implemetation
//--------------------------------------------------------------------------------------
// Entry action
	IF (me.StateMachine.intState<>me.StateMachine.intStateLastCycle) THEN
		me.StateMachine.intStateLastCycle := me.StateMachine.intState;
					
	END_IF


//--------------------------------------------------------------------------------------
// Cyclic action
	IF (me.StateMachine.intState=me.StateMachine.intStateLastCycle) THEN
	

		
		
		// State Change Condition
		IF SIf.par.pTblDecision = 0 THEN
			// SIf.Alm[2].strText := 'RUN not possible, no Hashtable';
			pfbAlarmCtrl^.setAlarm(CIf.Info.intCtrlId,2,0,ADR(SIf.Alm),E_AlmState.RST,CIf.Job.eMe_ActivAlmClass);	
			me.StateMachine.intStateNext := cSTA_ERROR;
		ELSE
			me.StateMachine.intStateNext := cSTA_RUN;		
		END_IF
	END_IF




//--------------------------------------------------------------------------------------
// Exit action
	IF (me.StateMachine.intState<>me.StateMachine.intStateNext) THEN
		;
	END_IF
END_METHOD

METHOD PROTECTED sta_STOP : BOOL
// state implemetation
//--------------------------------------------------------------------------------------
// Entry action
	IF (me.StateMachine.intState<>me.StateMachine.intStateLastCycle) THEN
		me.StateMachine.intStateLastCycle := me.StateMachine.intState;
		
	END_IF


//--------------------------------------------------------------------------------------
// Cyclic action
	IF (me.StateMachine.intState=me.StateMachine.intStateLastCycle) THEN
	
		
		// State Change Condition
		IF (me.intCmd=JUN_CmdState.cCMD_RELEASE) THEN 
			me.StateMachine.intStateNext := JUN_CmdState.cSTA_RELEASEBusy;
		ELSIF(me.intCmd=JUN_CmdState.cCMD_RELEASE_ALL) THEN
			me.StateMachine.intStateNext := JUN_CmdState.cSTA_RELEASE_ALLBusy;
		ELSIF (me.intCmd=cCMD_RUN) THEN
			me.StateMachine.intStateNext := cSTA_RUNBusy;
		END_IF
	END_IF




//--------------------------------------------------------------------------------------
// Exit action
	IF (me.StateMachine.intState<>me.StateMachine.intStateNext) THEN
		;
	END_IF
END_METHOD

METHOD PROTECTED sta_STOPBusy : BOOL
// state implemetation
//--------------------------------------------------------------------------------------
// Entry action
	IF (me.StateMachine.intState<>me.StateMachine.intStateLastCycle) THEN
		me.StateMachine.intStateLastCycle := me.StateMachine.intState;

	END_IF


//--------------------------------------------------------------------------------------
// Cyclic action
	IF (me.StateMachine.intState=me.StateMachine.intStateLastCycle) THEN

		// Simulation
		
		//no change action
		SIf.Out.bolOpen.intern := FALSE;
		
		// State Change Condition
		IF (me.StateMachine.udiTimeInState_ms > SIf.Par.udiCloseTime_ms) THEN
			me.StateMachine.intStateNext := cSTA_STOP;
		END_IF
	END_IF




//--------------------------------------------------------------------------------------
// Exit action
	IF (me.StateMachine.intState<>me.StateMachine.intStateNext) THEN
		;
	END_IF
END_METHOD

METHOD PROTECTED StateMachine : BOOL
SUPER^.StateMachine();

// main statemachine of base controller
CASE me.StateMachine.intState OF
    cSTA_RUNBusy: 
        THIS^.sta_RUNBusy();
    cSTA_RUN: 
        THIS^.sta_RUN();
     cSTA_STOPBusy: 
        THIS^.sta_STOPBusy();
    cSTA_STOP: 
        THIS^.sta_STOP();
    JUN_CmdState.cSTA_RELEASE_ALLBusy: 
        THIS^.sta_RELEASE_ALLBusy();
    JUN_CmdState.cSTA_RELEASE_ALL: 
        THIS^.sta_RELEASE_ALL();
    JUN_CmdState.cSTA_RELEASEBusy: 
        THIS^.sta_RELEASEBusy();
    JUN_CmdState.cSTA_RELEASE: 
        THIS^.sta_RELEASE();
END_CASE;
END_METHOD

END_FUNCTION_BLOCK

// POUs/Controller/Lvl0/LAI (Labler Interface)/FB_LAI
FUNCTION_BLOCK FB_LAI EXTENDS FB_CtrlBase
VAR_INPUT
	In_bolReady: BOOL;
	In_bolNoError: BOOL;
	In_bolLowMaterial: BOOL;
	/// Feedback from Labler -> Labeling finished
	In_bolJobFinished: BOOL;
	In_bolCylInPosition: BOOL;
	In_bolErrLabel: BOOL;
	In_bolErrPrinter: BOOL;
	In_bolErrDrive: BOOL;
	In_bolErrCylinder: BOOL;
END_VAR
VAR_OUTPUT
	/// Enable labler in automatic mode
	Out_bolAutomaticOn: BOOL;
	/// Info to labler, product in position. Labler execute job with signal = TRUE 
	Out_bolProductInPos: BOOL;
END_VAR
VAR
	/// cmd from LineControl indicating hanger is in clamping position (inclusive reclamp) and ready for process step
	bolCMD_PRODUCT_IN_POSITION: BOOL;
	/// Specific interface struct for public access
	SIf: T_Ctrl_SIf_LAI;
	/// Loop variable
	intI: INT;
END_VAR
VAR CONSTANT
	cSTA_SUB_WAIT_FOR_HANGER: INT := 300;
	cSTA_SUB_EXECUTE_PRINT_JOB: INT := 301;
	cSTA_SUB_WAIT_JOB_FINISHED: INT := 302;
END_VAR

(*__________________________________________________________________________________________________
¦	
¦	Vistaprint Schweiz GmbH
¦	CH - 8401 Winterthur
¦
¦	www.vistaprint.ch - info@vistaprint.ch
¦___________________________________________________________________________________________________

Function desription:
Interface to external Labler
Labler gets the data directly from the Line Controller
This interface only checks the state of the Labler and set errormessages


History:
Version		Date			Author		Comment
---------------------------------------------------------------------------------------------------
0.00.1		11.09.2013		AVME/PRE	Start history
0.00.2		19.09.2013		AVME/PRE	Implement new Base Concept
0.00.3		02.10.2013		AVME/MRU	New simulation time in RUN and RUNBusy
0.00.4		08.10.2013		VP/RE		Bug fixes, tested during FAT
0.00.5		21.10.2013		AVME/MRU	Some changes for Simulation
0.00.6		04.12.2013		AVME/DSC	Some changes for Simulation
___________________________________________________________________________________________________*)


IF (me.bolActivate) THEN // cyclic call enabled
	IF (CIf.Info.bolInitDone=FALSE) THEN // first cycle -> init
		CtrlInit();
		CIf.Info.bolInitDone := TRUE;
	ELSE
		CycleStartDuty();
	
		Always();
		
		StateMachine();
		
		CycleEndDuty();
	END_IF
END_IF;

METHOD PROTECTED Always : BOOL
SUPER^.Always();

IF (me.StateMachine.intState<>cSTA_SINGLE_ANSWER) THEN
	;
END_IF

// overrule error always from base -> no EOFF State!! in EOFF go to OFF
IF (me.StateMachine.intStateNext = cSTA_EOFFBusy) THEN
	IF (me.StateMachine.intState=cSTA_OFF) THEN
		me.StateMachine.intStateNext := cSTA_OFF;
	ELSE // stay in OFF
		me.StateMachine.intStateNext := cSTA_OFFBusy;
	END_IF
END_IF

// Conditions Always
IF (((me.Alarm.eActivAlmClass=E_AlmClass.EOFF) OR (me.Alarm.eActivAlmClass=E_AlmClass.OFF) OR (me.intCmd=cCMD_OFF))
		 AND (me.StateMachine.intState<>cSTA_ERROR) AND (me.StateMachine.intState<>cSTA_ERRORQuit) AND
		(me.StateMachine.intState<>cSTA_OFF) AND (me.StateMachine.intState<>cSTA_OFFBusy)) THEN
	// alarm evt EOFF, OFF or cmd off
	me.StateMachine.intStateNext := cSTA_OFFBusy;
END_IF
END_METHOD

METHOD FB_init : BOOL
VAR_INPUT
	///if TRUE, the retain variables are initialized (warm start / cold start)
	bInitRetains: BOOL;
	///if TRUE, the instance afterwards gets moved into the copy code (online change)
	bInCopyCode: BOOL;
END_VAR
VAR
	ii: UINT;
END_VAR
//------------------------------------------------------------------------------------------------------------------------
// to manually change in new FUB implementation!!!
// define valid commands for this controller
FOR ii:= 0 TO (SIZEOF(CIf.Job.aCmdList)/SIZEOF(CIf.Job.aCmdList[0])-1) BY 1 DO
	IF (CIf.Job.aCmdList[ii].intCmd=cCMD_INITIALIZED) THEN
		// found first empty array element
		EXIT;
	END_IF
END_FOR

CIf.Job.aCmdList[ii].intCmd := cCMD_RUN;
CIf.Job.aCmdList[ii].strName := 'Run'; 
CIf.Job.aCmdList[ii].bolAvailable := TRUE;
ii := ii +1;

// set name of class/typ
CIf.Info.strType := 'FB_LAI'; 

// set alarm class
SIf.Alm[1].eAlmClass := E_AlmClass.INFO;
SIf.Alm[1].strText := 'Labler not ready'; 
SIf.Alm[2].eAlmClass := E_AlmClass.OFF;
SIf.Alm[2].strText := 'General fault active';
SIf.Alm[3].eAlmClass := E_AlmClass.OFF;
SIf.Alm[3].strText := 'Label error'; 
SIf.Alm[4].eAlmClass := E_AlmClass.OFF;
SIf.Alm[4].strText := 'Printer error';
SIf.Alm[5].eAlmClass := E_AlmClass.OFF;
SIf.Alm[5].strText := 'Drive error';
SIf.Alm[6].eAlmClass := E_AlmClass.OFF;
SIf.Alm[6].strText := 'Cylinder error'; 
SIf.Alm[7].eAlmClass := E_AlmClass.OFF;
SIf.Alm[7].strText := 'Error 6';

//*******************************************************************************
// initial values
//*******************************************************************************

// software configuration
CIf.SwCfg.bolExist := TRUE;
CIf.SwCfg.bolSimulation := FALSE;

// parmeter
SIf.Par.udi_TimeoutReady_ms := 10000;
SIf.Par.udi_SimReady_ms := SIf.Par.udi_TimeoutReady_ms/2;
SIf.Par.udi_Finished_ms := 10000;
END_METHOD

METHOD PROTECTED getCmdState : STRING
VAR_INPUT
	intCmdState: INT;
	bolState: BOOL;
END_VAR
getCmdState := SUPER^.getCmdState(intCmdState:=intCmdState,bolState:=bolState); // get global/base defined cmds/states
IF (getCmdState='') THEN // global not defined get local
	// get string cmd/state string information in runtime
	IF (bolState=FALSE) THEN
		// cmd's
		CASE intCmdState OF
		END_CASE;
	ELSE
	
	// states
		CASE intCmdState OF		
			// SUB States
			cSTA_SUB_WAIT_FOR_HANGER:
				getCmdState := 'cSTA_SUB_WAIT_FOR_HANGER';
			cSTA_SUB_EXECUTE_PRINT_JOB:
				getCmdState := 'cSTA_SUB_EXECUTE_PRINT_JOB';
			cSTA_SUB_WAIT_JOB_FINISHED:
				getCmdState := 'cSTA_SUB_WAIT_JOB_FINISHED';										
		END_CASE;
	END_IF
END_IF
END_METHOD

METHOD getCtrlSIf : POINTER TO T_Ctrl_SIf_LAI
getCtrlSIf := ADR(SIf);
END_METHOD

METHOD PROTECTED IoInBridge : BOOL
// digitale and analoge inputs read from hardware or forcing

SIf.In.bolReady.map := THIS^.In_bolReady;
SIf.In.bolNoError.map := THIS^.In_bolNoError;
SIf.In.bolLowMaterial.map := THIS^.In_bolLowMaterial;
SIf.In.bolJobFinished.map := THIS^.In_bolJobFinished;
SIf.In.bolCylInPosition.map := THIS^.In_bolCylInPosition;
SIf.In.bolErrLabel.map := THIS^.In_bolErrLabel;
SIf.In.bolErrPrinter.map := THIS^.In_bolErrPrinter;
SIf.In.bolErrDrive.map := THIS^.In_bolErrDrive;
SIf.In.bolErrCylinder.map := THIS^.In_bolErrCylinder;

IF (CIf.SwCfg.bolSimulation = FALSE) THEN	
	getInBol(CIf.Job.bolIoForce,ADR(SIf.In.bolReady));
	getInBol(CIf.Job.bolIoForce,ADR(SIf.In.bolNoError));
	getInBol(CIf.Job.bolIoForce,ADR(SIf.In.bolLowMaterial));
	getInBol(CIf.Job.bolIoForce,ADR(SIf.In.bolJobFinished));
	getInBol(CIf.Job.bolIoForce,ADR(SIf.In.bolCylInPosition));
	getInBol(CIf.Job.bolIoForce,ADR(SIf.In.bolErrLabel));
	getInBol(CIf.Job.bolIoForce,ADR(SIf.In.bolErrPrinter));
	getInBol(CIf.Job.bolIoForce,ADR(SIf.In.bolErrDrive));
	getInBol(CIf.Job.bolIoForce,ADR(SIf.In.bolErrCylinder));
	//ctrl.In.bol_PosSwitchBasicDefTyp.intern := getInBol(ctrl.ifc.Job.bol_Force ,ADR(ctrl.In.bol_PosSwitchBasicDefTyp);
ELSE
	//simulation of global IO
END_IF
END_METHOD

METHOD PROTECTED IoOutBridge : BOOL
// digitale and analoge inputs read from hardware or forcing
IF (CIf.SwCfg.bolSimulation = FALSE) THEN
	
	setOutBol(CIf.Job.bolIoForce ,ADR(SIf.Out.bolAutomaticOn));
	setOutBol(CIf.Job.bolIoForce ,ADR(SIf.Out.bolProductInPos));
	
	THIS^.Out_bolAutomaticOn := SIf.Out.bolAutomaticOn.map;
	THIS^.Out_bolProductInPos := SIf.Out.bolProductInPos.map;
	
END_IF
END_METHOD

METHOD PROTECTED sta_ERROR : BOOL
// state implemetation
//--------------------------------------------------------------------------------------
// Entry action
IF (me.StateMachine.intState<>me.StateMachine.intStateLastCycle) THEN
	me.StateMachine.intStateHistory := me.StateMachine.intStateLastCycle; // -> possibillity to go back to state before error
	me.StateMachine.intStateLastCycle := me.StateMachine.intState;
	;
END_IF

//--------------------------------------------------------------------------------------
// Cyclic action
	IF (me.StateMachine.intState=me.StateMachine.intStateLastCycle) THEN
		
		// Labler off
		SIf.Out.bolAutomaticOn.intern := FALSE;
		SIf.Out.bolProductInPos.intern := FALSE;

		// State Change Condition
		IF (CIf.Job.bolAlmReset = TRUE) THEN
			me.StateMachine.intStateNext := cSTA_ERRORQuit;
		END_IF
	END_IF

//--------------------------------------------------------------------------------------
// Exit action
	IF (me.StateMachine.intState<>me.StateMachine.intStateNext) THEN
		;
	END_IF
END_METHOD

METHOD PROTECTED sta_OFF : BOOL
// state implemetation
//--------------------------------------------------------------------------------------
// Entry action
	IF (me.StateMachine.intState<>me.StateMachine.intStateLastCycle) THEN
		me.StateMachine.intStateLastCycle := me.StateMachine.intState;
		
	END_IF

//--------------------------------------------------------------------------------------
// Cyclic action
	IF (me.StateMachine.intState=me.StateMachine.intStateLastCycle) THEN
		
		;
			
		// State Change Condition
		IF (me.intCmd=cCMD_RUN) THEN 
			me.StateMachine.intStateNext := cSTA_RUNBusy;
		END_IF
	END_IF

//--------------------------------------------------------------------------------------
// Exit action
	IF (me.StateMachine.intState<>me.StateMachine.intStateNext) THEN
		;
	END_IF
END_METHOD

METHOD PROTECTED sta_OFFBusy : BOOL
// state implemetation
//--------------------------------------------------------------------------------------
// Entry action
	IF (me.StateMachine.intState<>me.StateMachine.intStateLastCycle) THEN
		me.StateMachine.intStateLastCycle := me.StateMachine.intState;
		
	END_IF

//--------------------------------------------------------------------------------------
// Cyclic action
	IF (me.StateMachine.intState=me.StateMachine.intStateLastCycle) THEN
		
		// Labler off
		SIf.Out.bolAutomaticOn.intern := FALSE;
		SIf.Out.bolProductInPos.intern := FALSE;
				
		// State Change Condition
		IF (TRUE) THEN
			me.StateMachine.intStateNext := cSTA_OFF;
		END_IF
	END_IF

//--------------------------------------------------------------------------------------
// Exit action
	IF (me.StateMachine.intState<>me.StateMachine.intStateNext) THEN
		;
	END_IF
END_METHOD

METHOD PROTECTED sta_RUN : BOOL
// state implemetation
//--------------------------------------------------------------------------------------
// Entry action
	IF (me.StateMachine.intState<>me.StateMachine.intStateLastCycle) THEN
		me.StateMachine.intStateLastCycle := me.StateMachine.intState;
		
		fbSimulationTimer.IN := FALSE;
		fbSimulationTimer.PT := UDINT_TO_TIME(SIf.Par.udi_SimReady_ms ); // Divide 2 because of toggle, every 
		fbSimulationTimer(); // set time/reset timer
		fbSimulationTimer.IN := TRUE; // start timer
		
		// Initialize sub state machine
		me.SubStateMachine.intState:= cSTA_SUB_WAIT_FOR_HANGER; 
		me.SubStateMachine.intStateNext:= cSTA_SUB_WAIT_FOR_HANGER;
		SIf.Cur.bolJobFinished:= TRUE;
		
	END_IF


//--------------------------------------------------------------------------------------
// Cyclic action
	IF (me.StateMachine.intState=me.StateMachine.intStateLastCycle) THEN
		
		// Simulation
		IF (CIf.SwCfg.bolSimulation) THEN
			fbSimulationTimer(); // simulation time
			IF (fbSimulationTimer.Q) THEN
				SIf.In.bolJobFinished.intern := NOT SIf.In.bolJobFinished.intern; // toggle pulse
				fbSimulationTimer.IN := FALSE;
			ELSE
				fbSimulationTimer.IN := TRUE;
			END_IF
			SIf.In.bolNoError.intern := TRUE;	// Simulate no errror
		END_IF
		
		//---------------------------------------------------------
		// Check Alarms from Labler
		//---------------------------------------------------------
	
		IF SIf.In.bolNoError.intern = FALSE THEN
			// Set Alarm: SIf.Alm[2].strText := 'General fault active';
			pfbAlarmCtrl^.setAlarm(CIf.Info.intCtrlId,2,0,ADR(SIf.Alm),E_AlmState.RST,CIf.Job.eMe_ActivAlmClass);	
			me.StateMachine.intStateNext :=  cSTA_ERROR;	
		END_IF
		
		IF SIf.In.bolErrLabel.intern = TRUE THEN
			// Set Alarm: SIf.Alm[3].strText := 'Label error'; 
			pfbAlarmCtrl^.setAlarm(CIf.Info.intCtrlId,3,0,ADR(SIf.Alm),E_AlmState.RST,CIf.Job.eMe_ActivAlmClass);
			me.StateMachine.intStateNext :=  cSTA_ERROR;		
		END_IF
				
		IF SIf.In.bolErrPrinter.intern = TRUE THEN
			// Set Alarm: SIf.Alm[4].strText := 'Printer error';
			pfbAlarmCtrl^.setAlarm(CIf.Info.intCtrlId,4,0,ADR(SIf.Alm),E_AlmState.RST,CIf.Job.eMe_ActivAlmClass);
			me.StateMachine.intStateNext :=  cSTA_ERROR;			
		END_IF
		
		IF SIf.In.bolErrDrive.intern = TRUE THEN
			// Set Alarm: SIf.Alm[5].strText := 'Drive error';
			pfbAlarmCtrl^.setAlarm(CIf.Info.intCtrlId,5,0,ADR(SIf.Alm),E_AlmState.RST,CIf.Job.eMe_ActivAlmClass);
			me.StateMachine.intStateNext :=  cSTA_ERROR;			
		END_IF
		
		IF SIf.In.bolErrCylinder.intern = TRUE THEN
			// Set Alarm: SIf.Alm[6].strText := 'Cylinder error'; 
			pfbAlarmCtrl^.setAlarm(CIf.Info.intCtrlId,6,0,ADR(SIf.Alm),E_AlmState.RST,CIf.Job.eMe_ActivAlmClass);
			me.StateMachine.intStateNext :=  cSTA_ERROR;			
		END_IF
	
	
		//--------------------------------------------------------------------------------------
		// sub state machine for Handshake between line control and labler
		//--------------------------------------------------------------------------------------
		CASE me.SubStateMachine.intState OF
		
			cSTA_SUB_WAIT_FOR_HANGER:
			
				// Signal from line control
				IF (bolCMD_PRODUCT_IN_POSITION = TRUE) THEN
					bolCMD_PRODUCT_IN_POSITION := FALSE;
					SIf.Cur.bolJobFinished := FALSE;
					me.SubStateMachine.intStateNext := cSTA_SUB_EXECUTE_PRINT_JOB;
				END_IF
	
			cSTA_SUB_EXECUTE_PRINT_JOB:
					
				// State Change Condition
				//IF (SIf.In.bolJobFinished.intern=FALSE) AND (SIf.In.bolCylInPosition.intern=TRUE) THEN
					// Info to labler, product in position. Labler execute print job!
					SIf.Out.bolProductInPos.intern := TRUE;
					me.SubStateMachine.intStateNext := cSTA_SUB_WAIT_JOB_FINISHED;
				//END_IF

			cSTA_SUB_WAIT_JOB_FINISHED:
	
				// State Change Condition
				IF (SIf.In.bolJobFinished.intern=TRUE) AND (SIf.In.bolCylInPosition.intern=TRUE) THEN
					SIf.Out.bolProductInPos.intern:= FALSE;
					SIf.Cur.bolJobFinished:= TRUE;
					me.SubStateMachine.intStateNext := cSTA_SUB_WAIT_FOR_HANGER;
				END_IF		
					
		END_CASE
			

		// State Change Condition
		IF (SIf.In.bolReady.intern = FALSE) THEN 
			me.StateMachine.intStateNext := cSTA_ERROR;
		END_IF
	
	END_IF
//--------------------------------------------------------------------------------------
// Exit action
	IF (me.StateMachine.intState<>me.StateMachine.intStateNext) THEN
		;
	END_IF
END_METHOD

METHOD PROTECTED sta_RUNBusy : BOOL
// state implemetation
//--------------------------------------------------------------------------------------
// Entry action
	IF (me.StateMachine.intState<>me.StateMachine.intStateLastCycle) THEN
		me.StateMachine.intStateLastCycle := me.StateMachine.intState;

		fbSimulationTimer.IN := FALSE;
		fbSimulationTimer.PT := UDINT_TO_TIME(SIf.Par.udi_SimReady_ms); // Divide 2 because of toggle, every 
		fbSimulationTimer(); // set time/reset timer
		fbSimulationTimer.IN := TRUE; // start timer
		
	END_IF

//--------------------------------------------------------------------------------------
// Cyclic action
	IF (me.StateMachine.intState=me.StateMachine.intStateLastCycle) THEN

		// Simulation
		IF (CIf.SwCfg.bolSimulation) THEN
			fbSimulationTimer(); // simulation time
			IF (fbSimulationTimer.Q) THEN		
				SIf.In.bolReady.intern := TRUE;
			END_IF
			SIf.In.bolCylInPosition.intern := TRUE;	// Simulate Cyl in Position
		END_IF
		
		// Labler on
		SIf.Out.bolAutomaticOn.intern := TRUE;
				
		// State Change Condition
		IF (me.StateMachine.udiTimeInState_ms>SIf.Par.udi_TimeoutReady_ms) THEN
			// Set Alarm: SIf.Alm[1].strText := 'Labler not ready';
			pfbAlarmCtrl^.setAlarm(CIf.Info.intCtrlId,1,0,ADR(SIf.Alm),E_AlmState.RST,CIf.Job.eMe_ActivAlmClass);
			me.StateMachine.intStateNext := cSTA_ERROR;
		ELSIF (SIf.In.bolReady.intern = TRUE) AND (SIf.In.bolCylInPosition.intern = TRUE) THEN
			me.StateMachine.intStateNext := cSTA_RUN;
		END_IF
	END_IF

//--------------------------------------------------------------------------------------
// Exit action
	IF (me.StateMachine.intState<>me.StateMachine.intStateNext) THEN
		;
	END_IF
END_METHOD

METHOD PROTECTED StateMachine : BOOL
SUPER^.StateMachine();

// main statemachine of base controller
CASE me.StateMachine.intState OF
    cSTA_RUNBusy: 
        THIS^.sta_RUNBusy();
    cSTA_RUN: 
        THIS^.sta_RUN();
END_CASE;
END_METHOD

END_FUNCTION_BLOCK

// POUs/Controller/Lvl0/PLS (PickToLight System)/FB_PLS
FUNCTION_BLOCK FB_PLS EXTENDS FB_CtrlBase
VAR_OUTPUT
	Out_Lights: ARRAY[0..MAX_SKUS] OF BYTE;
END_VAR
VAR
	/// Specific interface struct for public access
	SIf: T_Ctrl_SIf_PLS;
	iBlinkLights: ARRAY[0..MAX_SKUS] OF BYTE;
	toggle: BOOL;
	blinkTimer: TON;
	i: INT;
END_VAR

(*__________________________________________________________________________________________________
¦	
¦	Vistaprint Schweiz GmbH
¦	CH - 8401 Winterthur
¦
¦	www.vistaprint.ch - info@vistaprint.ch
¦___________________________________________________________________________________________________

Function desription:
Pick to light system


History:
Version		Date			Author		Comment
---------------------------------------------------------------------------------------------------
0.00.1		02.07.2013		VP/RE		Start history
0.00.2		16.12.2013		AVME/MRU	Add Method Always


___________________________________________________________________________________________________*)


IF (me.bolActivate) THEN // cyclic call enabled
	IF (CIf.Info.bolInitDone=FALSE) THEN // first cycle -> init
		CtrlInit();
		CIf.Info.bolInitDone := TRUE;
	ELSE
		CycleStartDuty();
	
		Always();
		
		StateMachine();
		
		CycleEndDuty();
	END_IF
END_IF;

METHOD PROTECTED Always : BOOL
SUPER^.Always();

IF (me.StateMachine.intState<>cSTA_SINGLE_ANSWER) THEN
	
	;
	
END_IF

// ----------------------------------------------------------------------------------
// Conditions Always
// overrule error always from base -> no EOFF State!! in EOFF go to OFF
IF (me.StateMachine.intStateNext = cSTA_EOFFBusy) THEN
	IF (me.StateMachine.intState=cSTA_OFF) THEN
		me.StateMachine.intStateNext := cSTA_OFF;
	ELSE // stay in OFF
		me.StateMachine.intStateNext := cSTA_OFFBusy;
	END_IF
END_IF
END_METHOD

METHOD PROTECTED CtrlInit : BOOL
SUPER^.CtrlInit();
END_METHOD

METHOD FB_init : BOOL
VAR_INPUT
	///if TRUE, the retain variables are initialized (warm start / cold start)
	bInitRetains: BOOL;
	///if TRUE, the instance afterwards gets moved into the copy code (online change)
	bInCopyCode: BOOL;
END_VAR
VAR
	ii: UINT;
END_VAR
//------------------------------------------------------------------------------------------------------------------------
// to manually change in new FUB implementation!!!
// define valid commands for this controller
FOR ii:= 0 TO (SIZEOF(CIf.Job.aCmdList)/SIZEOF(CIf.Job.aCmdList[0])-1) BY 1 DO
	IF (CIf.Job.aCmdList[ii].intCmd=cCMD_INITIALIZED) THEN
		// found first empty array element
		EXIT;
	END_IF
END_FOR
//CIf.Job.aCmdList[ii].intCmd := cCMD_RUN;
//CIf.Job.aCmdList[ii].strName := 'Run'; 
//CIf.Job.aCmdList[ii].bolAvailable := TRUE;
//ii := ii +1;
//CIf.Job.aCmdList[ii].intCmd := cCMD_RETRACT;
//CIf.Job.aCmdList[ii].strName := 'Retract';
//CIf.Job.aCmdList[ii].bolAvailable := TRUE;

// set name of class/typ
CIf.Info.strType := 'FB_PLS'; 

// set alarm class
//SIf.Alm[1].eAlmClass := E_AlmClass.TSTOP;
//SIf.Alm[1].strText := 'sensor retract always on'; 


//*******************************************************************************
// initial values
//*******************************************************************************

// software configuration
CIf.SwCfg.bolExist := TRUE;
CIf.SwCfg.bolSimulation := FALSE;

// parmeter
//SIf.Par.udiHangerLoadingTime_ms := 800;

// actual values
SIf.Cur.dinCounter := 0;
END_METHOD

METHOD PROTECTED getCmdState : STRING
VAR_INPUT
	intCmdState: INT;
	bolState: BOOL;
END_VAR
getCmdState := SUPER^.getCmdState(intCmdState:=intCmdState,bolState:=bolState); // get global/base defined cmds/states

IF (getCmdState='') THEN // global not defined get local
	// get string cmd/state string information in runtime
	IF (bolState=FALSE) THEN
		// cmd's
		CASE intCmdState OF
			//cCMD_RETRACT: 
			//	getCmdState := 'cCMD_RETRACT';
		END_CASE;
	ELSE
	
	// cmd's
		CASE intCmdState OF
			//cSTA_RETRACTBusy: 
			//	getCmdState := 'cSTA_RETRACTBusy';
			//cSTA_RETRACT: 
			//	getCmdState := 'cSTA_RETRACT';
		END_CASE;
	END_IF
END_IF
END_METHOD

METHOD getCtrlSIf : POINTER TO T_Ctrl_SIf_PLS
getCtrlSIf := ADR(SIf);
END_METHOD

METHOD PROTECTED IoInBridge : BOOL
// digitale and analoge inputs read from hardware or forcing
//SIf.In.bolGiveNextHangerSensor.map := THIS^.In_GiveNextHangerSensor;

IF (CIf.SwCfg.bolSimulation = FALSE) THEN
	//getInBol(CIf.Job.bolIoForce,ADR(SIf.In.bolGiveNextHangerSensor));
	
ELSE
	//simulation of global IO
END_IF
END_METHOD

METHOD PROTECTED IoOutBridge : BOOL
VAR
	bolSwitchValvesOff: BOOL;
END_VAR
// digitale and analoge inputs read from hardware or forcing
IF (CIf.SwCfg.bolSimulation = FALSE) THEN
	//setOutBol(CIf.Job.bolIoForce ,ADR(SIf.Out.bolClamping));
	
	//THIS^.Out_Clamping := SIf.Out.bolClamping.map;
END_IF
END_METHOD

METHOD PROTECTED sta_ERROR : BOOL
// state implemetation
//--------------------------------------------------------------------------------------
// Entry action
	IF (me.StateMachine.intState<>me.StateMachine.intStateLastCycle) THEN
		me.StateMachine.intStateHistory := me.StateMachine.intStateLastCycle; // -> possibillity to go back to state before error
		me.StateMachine.intStateLastCycle := me.StateMachine.intState;
		
	END_IF


//--------------------------------------------------------------------------------------
// Cyclic action
	IF (me.StateMachine.intState=me.StateMachine.intStateLastCycle) THEN
		
		;
		
		
		// State Change Condition
		IF (CIf.Job.bolAlmReset = TRUE) THEN
			me.StateMachine.intStateNext := cSTA_ERRORQuit;
		END_IF
	END_IF




//--------------------------------------------------------------------------------------
// Exit action
	IF (me.StateMachine.intState<>me.StateMachine.intStateNext) THEN
		;
	END_IF
END_METHOD

METHOD PROTECTED sta_ERRORQuit : BOOL
// state implemetation
//--------------------------------------------------------------------------------------
// Entry action
	IF (me.StateMachine.intState<>me.StateMachine.intStateLastCycle) THEN
		me.StateMachine.intStateLastCycle := me.StateMachine.intState;
		
	END_IF


//--------------------------------------------------------------------------------------
// Cyclic action
	IF (me.StateMachine.intState=me.StateMachine.intStateLastCycle) THEN
		
		;
		// evtl. wait time if reset of device is necessary and then decide to go to states or ERROR state
		IF (CIf.Job.bolAlmReset = TRUE) THEN
			CIf.Job.eMe_ActivAlmClass := E_AlmClass.NONE; // reset feedback channel for parent
			CIf.Job.bolAlmReset := FALSE;
		END_IF
		
		// State Change Condition
		IF (CIf.Job.bolAlmReset = FALSE) THEN
			IF (me.StateMachine.intStateHistory<=cSTA_PON) THEN
				me.StateMachine.intStateNext := cSTA_PONBusy;
			ELSIF(me.intCmd=cCMD_OFF) THEN
				me.StateMachine.intStateNext := cSTA_OFFBusy;
			ELSIF(me.intCmd=cCMD_STOP) THEN
				me.StateMachine.intStateNext := cSTA_STOPBusy;
			ELSIF(me.intCmd=cCMD_RUN) THEN
				me.StateMachine.intStateNext := cSTA_RUNBusy;
			END_IF
		END_IF
	END_IF




//--------------------------------------------------------------------------------------
// Exit action
	IF (me.StateMachine.intState<>me.StateMachine.intStateNext) THEN
		;
	END_IF
END_METHOD

METHOD PROTECTED sta_OFF : BOOL
// state implemetation
//--------------------------------------------------------------------------------------
// Entry action
	IF (me.StateMachine.intState<>me.StateMachine.intStateLastCycle) THEN
		me.StateMachine.intStateLastCycle := me.StateMachine.intState;
		
	END_IF


//--------------------------------------------------------------------------------------
// Cyclic action
	IF (me.StateMachine.intState=me.StateMachine.intStateLastCycle) THEN
		
		;
		
		// State Change Condition
		IF (me.intCmd=cCMD_RUN) THEN
			me.StateMachine.intStateNext :=  cSTA_RUN;
		END_IF
	END_IF

//--------------------------------------------------------------------------------------
// Exit action
	IF (me.StateMachine.intState<>me.StateMachine.intStateNext) THEN
		;
	END_IF
END_METHOD

METHOD PROTECTED sta_RUN : BOOL
// state implemetation
//--------------------------------------------------------------------------------------
// Entry action
	IF (me.StateMachine.intState<>me.StateMachine.intStateLastCycle) THEN
		me.StateMachine.intStateLastCycle := me.StateMachine.intState;
		;
	END_IF

//--------------------------------------------------------------------------------------
// Cyclic action
IF (me.StateMachine.intState=me.StateMachine.intStateLastCycle) THEN	
	// light control
	blinkTimer(in := NOT(blinkTimer.Q), pt := T#500MS);

	IF blinkTimer.Q THEN
		toggle := NOT(toggle);
	END_IF
	
	FOR i := 0 TO MAX_SKUS - 1 DO
		IF iBlinkLights[i] > 0 THEN
			IF toggle THEN
				Out_Lights[i] := iBlinkLights[i];
			ELSE
				Out_Lights[i] := 0;
			END_IF
		END_IF
	END_FOR
	
	// State Change Condition
	// always in base -> OFF
	
END_IF	

//--------------------------------------------------------------------------------------
// Exit action
	IF (me.StateMachine.intState<>me.StateMachine.intStateNext) THEN
		;
	END_IF
END_METHOD

METHOD PROTECTED StateMachine : BOOL
SUPER^.StateMachine();

// main statemachine of base controller
CASE me.StateMachine.intState OF
	 cSTA_RUN: 
        THIS^.sta_RUN();
END_CASE;
END_METHOD

END_FUNCTION_BLOCK

// POUs/Controller/Lvl0/STB (Stopper buffer)/FB_STB
FUNCTION_BLOCK FB_STB EXTENDS FB_CtrlBase IMPLEMENTS IBuffer
VAR_INPUT
	/// Sensor hanger detected
	In_bolHangerDetected: BOOL;
	/// Buffer full sensor
	In_bolBufferFull: BOOL;
	/// DecrementCounter Sensor (option)
	In_bolDecrementCounter: BOOL;
END_VAR
VAR_OUTPUT
	/// if bolRetract2 is not used  = 1 -> second pin up first pin (inlet) down
	Out_bolRetract: BOOL;
	/// = 1 -> second pin down (outlet)
	Out_bolRetract2: BOOL;
END_VAR
VAR
	/// Specific interface struct for public access
	SIf: T_Ctrl_SIf_STB;
	/// Internal Variables
	bolHangerDetected: BOOL;
	dinNumOfHangersToRelease: DINT;
	dinSetNumOfHangersToRelease: DINT;
	bolSensorBufferFull: BOOL;
	bolSensorHangerDetected: BOOL;
	bolBufferFullOld: BOOL;
	bolBufferFullSigCountOld: BOOL;
	/// Shadow copy of SIf.In.bolDecrementCounter.intern
	bolDecrementCountOld: BOOL;
	bolSignalForPosLostMonitoring: BOOL;
	bolSignalForPosLostMonitoringOld: BOOL;
	uinPosEdgeCounter: UINT;
	bolErrorPosLost: BOOL;
	fbTimerBufferFullSignal: TON;
	fbTimerHangerDetecSignal: TON;
	fbTimerHangerDeleteNoDetected: TON;
	/// Var. used for simulation
	bolRESimHangerIn: BOOL;
	/// Rising Edge Hanger go out
	bolRESimHangerOut: BOOL;
	/// Var. used for decrementing with sensor
	bolWaitForDecrement: BOOL;
	/// Copy of Output
	bolRetractOld: BOOL;
END_VAR
VAR CONSTANT
	/// sub States for RELEASE_ALL Function
	cSTA_SUB_INITIALIZED: INT := 500;
	cSTA_SUB_HANGER_PASSING: INT := 502;
	cSTA_SUB_HANGER_PASSED: INT := 504;
	cSTA_SUB_FINISHED: INT := 506;
END_VAR

(*__________________________________________________________________________________________________
¦	
¦	Vistaprint Schweiz GmbH
¦	CH - 8401 Winterthur
¦
¦	www.vistaprint.ch - info@vistaprint.ch
¦___________________________________________________________________________________________________

Function desription:
The stopper buffer controller let pass hanger(s) with every pulse (retract/extend) of the pneumatic cylinder.
This controller can be used for the following units: Separator, Double stopper and Single stopper.

Note:  With the given sensors it's not possible to detect exactly one hanger per sensor pulse to inc. the number of hangers in buffer.
       Means that all calculated values ​​are only approximate.

History:
Version		Date			Author		Comment
---------------------------------------------------------------------------------------------------
0.00.1		22.08.2013		AVME/PRE	Start history
0.00.2		29.08.2013		AVME/DSC	Integration of all separator basic functionalities
0.00.3		30.08.2013		AVME/DSC	Integration monitoring cylinder position lost in state STOP.
0.00.4      09.09.2013      AVME/DSC    Generate signal "hanger detected". In case if only buffer full sensor exist, 
										use number of hangers to generate hanger detection signal.
										Renaming FUB "FB_SEP" to "FB_STB". Decided by Rolf and PRE.
0.00.5		19.09.2013		AVME/PRE	Limit Counter to max capacity if higher as max capacity
0.00.6		19.09.2013		AVME/PRE	Implement new Base Concept
0.00.7		26.09.2013		AVME/KVO	- Add new output for douplestopper with two valves
										- Add new config bolReleaseAllNonPulse -> to release all over time 
											-> new par udiReleaseAllTime_ms: UDINT;
										- calculation of hangers corrected
										- if hanger dtedction sensor detects a hanger and buffer is 0 -> set 1 always
										-  max number of hangers detected in STOP if bolCylPosLostMonitoring activated until an error occures
											uinMaxNumOfHangers_PosMonitoring
										- info buffer full and hanger detected removed - not necessary
0.00.8		27.09.2013		AVME/DSC	Modification for error condition of hanger position lost monitoring.										
0.00.9		02.10.2013		AVME/DSC	Modification set number of hangers in buffer to max. capacity if buffer full signal detected.
0.00.10		07.10.2013		AVME/DSC    Modification in always action. If buffer full detected, number of hangers in buffer must be always set to max. capacity.
0.00.11		09.10.2013		VP/RE		Only decrease dinNumOfHangersInBuffer when is NOT full (but only if full sensor is available)
0.00.12		07.11.2013		AVME/MRU	Add debounced inputs and configuration with bolHasDecrementSensor
0.00.13		03.12.2013		AVME/MRU	Add MaxCapacity / NumOfHangers properties
0.00.14		12.12.2013		AVME/MRU	Bug fixed with decrement sensor, Min. Limit of dinNumOfHangersInBuffer = 0;
										Add bolDisableBufferDelete for preventing deleting buffer count 
0.00.15		17.12.2013		AVME/MRU	sta_Release_AllBusy Buffermode=0, Bug fixed
										Code review, some comments changed
0.00.16		10.01.2014		AVME/MRU	Bugzilla ID 55: Limitation of dinNumOfHangersInBuffer reworked
										Bug in Simulation resolved
0.00.17		13.01.2014		AVME/MRU	Bugzilla ID 03: BufferFull for LineControl added
___________________________________________________________________________________________*)


IF (me.bolActivate) THEN // cyclic call enabled
	IF (CIf.Info.bolInitDone=FALSE) THEN // first cycle -> init
		CtrlInit();
		CIf.Info.bolInitDone := TRUE;
	ELSE
		CycleStartDuty();
	
		Always();
		
		StateMachine();
		
		CycleEndDuty();
	END_IF
END_IF;

METHOD PROTECTED Always : BOOL
IF (me.bolChangeBackToAUTO=TRUE) THEN // switch mode to automatic switch off controller
	//me.StateMachine.intStateNext := cSTA_OFFBusy;
	me.bolChangeBackToAUTO := FALSE; // for cylinder no change to off when switch to automatic!!
END_IF

SUPER^.Always();

// ----------------------------------------------------------------------------------
// cyclic actions outside of statemachine
IF (me.StateMachine.intState<>cSTA_SINGLE_ANSWER) THEN
	//////////////////
	// Simulation
	IF (CIf.SwCfg.bolSimulation) THEN
		fbSimulationTimer(); // set time/reset timer
		
		// Simulate Hanger is coming into the stopper
		IF (SIf.Cfg.bolHasBufferFullSensor = TRUE) AND (SIf.Cfg.bolHasHangerDetection = TRUE) THEN 
			IF (SIf.In.bolBufferFull.intern = TRUE) AND (bolRESimHangerIn = FALSE) THEN
				SIf.In.bolHangerDetected.intern := TRUE;
				bolRESimHangerIn := TRUE;
			ELSIF (SIf.In.bolBufferFull.intern = FALSE) AND (bolRESimHangerIn = TRUE) THEN
				bolRESimHangerIn := FALSE;				
			END_IF
		END_IF
		// Use number of hangers to generate buffer full signal
		IF (SIf.Cur.dinNumOfHangersInBuffer >= SIf.Cfg.dinMaxCapacity) THEN
			SIf.In.bolBufferFull.intern := TRUE;
		ELSIF ((SIf.In.bolBufferFull.intern = TRUE) AND (SIf.Cur.dinNumOfHangersInBuffer < SIf.Cfg.dinMaxCapacity)) THEN
			SIf.In.bolBufferFull.intern := FALSE;
		END_IF
		// Use number of hangers to generate hanger detection signal
		IF (SIf.Cur.dinNumOfHangersInBuffer <= 0) AND (SIf.Out.bolRetract.intern = TRUE) THEN
			SIf.In.bolHangerDetected.intern := FALSE;
		END_IF

	END_IF  // END SIMULATION
	
	//--------------------------------------------------------------------
	// Generate info "buffer full" dependent the existing sensors
	// Input signal validation
	//--------------------------------------------------------------------
	// Prio 1. Always use the buffer full sensor if exists
	IF (SIf.Cfg.bolHasBufferFullSensor = TRUE) THEN
		// Use buffer full sensor signal
		bolSensorBufferFull:= SIf.In.bolBufferFull.intern;
	ELSE
		//Prio 2. Check if hanger detection sensor exists 
		IF (SIf.Cfg.bolHasHangerDetection = TRUE) THEN
			// Use hanger detected sensor for buffer full signal (e.g. Separator with only hanger detection sensor)
			bolSensorBufferFull:= SIf.In.bolHangerDetected.intern;
		ELSE
			//No sensor exist.
			bolSensorBufferFull:= FALSE;
		END_IF
	END_IF
		
	// Check sensor signal. Valid if TRUE for X-time
	fbTimerBufferFullSignal.IN := bolSensorBufferFull; // start timer
	fbTimerBufferFullSignal.PT := UDINT_TO_TIME(SIf.Par.udiSensorTime_ms);
	fbTimerBufferFullSignal();
	
	// Signal valid. Set info buffer full.
	IF (fbTimerBufferFullSignal.Q = TRUE) THEN
		SIf.Cur.bolBufferFull:= TRUE;
	ELSE
		SIf.Cur.bolBufferFull:= FALSE;
	END_IF
	
	
	//--------------------------------------------------------------------
	// Generate info "hanger detected" dependent the existing sensors
	// Input signal validation
	//--------------------------------------------------------------------
	
	// Prio 1. Always use the hanger detection sensor if exists
	IF (SIf.Cfg.bolHasHangerDetection = TRUE) THEN
		// Use hanger detection sensor signal
		bolSensorHangerDetected:= SIf.In.bolHangerDetected.intern;
	ELSE
		//Prio 2. Check if buffer full sensor exists 
		IF (SIf.Cfg.bolHasBufferFullSensor = TRUE) THEN
			// Use number of hangers to generate hanger detection signal
			IF (SIf.Cur.dinNumOfHangersInBuffer > 0) THEN
				bolSensorHangerDetected:= TRUE;
			ELSE
				bolSensorHangerDetected:= FALSE;
			END_IF
		ELSE
			//No sensor exist.
			bolSensorHangerDetected:= FALSE;
		END_IF
	END_IF
		
	// Check sensor signal. Valid if TRUE for X-time
	fbTimerHangerDetecSignal.IN := bolSensorHangerDetected; // start timer
	fbTimerHangerDetecSignal.PT := UDINT_TO_TIME(SIf.Par.udiSensorTime_ms);
	fbTimerHangerDetecSignal();
	
	// Signal valid. Set info buffer full.
	IF (fbTimerHangerDetecSignal.Q = TRUE) THEN
		SIf.Cur.bolHangerDetected:= TRUE;
	ELSE
		SIf.Cur.bolHangerDetected:= FALSE;
	END_IF
	
	
	//--------------------------------------------------------------------
	// Counter handling buffer level (number of hangers in buffer)
	//--------------------------------------------------------------------

	// Inc. number of hangers in buffer with every edge of sensor
	// Has buffer sensor ?
	IF (SIf.Cfg.bolHasBufferFullSensor = TRUE) THEN
		
		// Inc. only if the buffer is not full
		IF (SIf.Cur.bolBufferFull = FALSE) THEN
			
			// Detection positive edge from buffer full sensor
			IF ((SIf.In.bolBufferFull.intern <> bolBufferFullSigCountOld) AND (SIf.In.bolBufferFull.intern = TRUE)) THEN			
				// Inc. number of hangers in buffer by one!
				// Note: With the given sensors it's not possible to count exactly one hanger per sensor pulse.
				// e.g. On a slide, normally they pass more than one hanger the sensor position at the same time.		
				SIf.Cur.dinNumOfHangersInBuffer:= SIf.Cur.dinNumOfHangersInBuffer + 1;
			END_IF
			bolBufferFullSigCountOld:= SIf.In.bolBufferFull.intern;
			
		END_IF
	END_IF

	// Dec. number of hangers in buffer with every edge of sensor
	// Has decrement sensor ?
	IF (SIf.Cfg.bolHasDecrementSensor = TRUE) THEN
		
		// Check if hangers passed the decrement sensor, else decrement NumOfHangersPerPulse
		IF ((SIf.Out.bolRetract.intern <>bolRetractOld) AND (SIf.Out.bolRetract.intern = TRUE)) THEN
			IF (bolWaitForDecrement = FALSE) THEN
				bolWaitForDecrement := TRUE; // Start waiting
			ELSE // Counter is still waiting from the last cycle -> Maybe STB was physically empty
				SIf.Cur.dinNumOfHangersInBuffer := SIf.Cur.dinNumOfHangersInBuffer - SIf.Cfg.uinNumOfHangersPerPulse;
			END_IF		
		END_IF 
		bolRetractOld := SIf.Out.bolRetract.intern;		
			
		// Detection positive edge from decrement sensor
		IF ((SIf.In.bolDecrementCounter.intern <> bolDecrementCountOld) AND (SIf.In.bolDecrementCounter.intern = TRUE)) THEN			
			// Dec. number of hangers in buffer by one!
			// Note: With the given sensors it's not possible to count exactly one hanger per sensor pulse.
			// e.g. On a slide, normally they pass more than one hanger the sensor position at the same time.		
			SIf.Cur.dinNumOfHangersInBuffer:= SIf.Cur.dinNumOfHangersInBuffer - 1;
			bolWaitForDecrement := FALSE;	// reset waiting
		END_IF
		bolDecrementCountOld:= SIf.In.bolDecrementCounter.intern;
			
	END_IF

	// Reset NumOfHangersInBuffer if no Hanger detected
	// If Hanger detected, minimum 1 Hanger in Buffer
	IF (SIf.Cfg.bolHasHangerDetection = TRUE) THEN
		// With Sensor Hanger delete hanger counter if no hanger is detected
		// Check sensor signal. Valid if TRUE for X-time
		fbTimerHangerDeleteNoDetected.IN := NOT SIf.In.bolHangerDetected.intern; // start timer
		fbTimerHangerDeleteNoDetected.PT := UDINT_TO_TIME(SIf.Par.udiSensorTime_ms);
		fbTimerHangerDeleteNoDetected();
		
		// Signal valid. Set info buffer empty, if not prevented.
		IF ((fbTimerHangerDeleteNoDetected.Q = TRUE) AND (SIf.Cfg.bolDisableBufferDelete = FALSE)) THEN
			SIf.Cur.dinNumOfHangersInBuffer := 0;
		END_IF
		
		// sensor has at least one hanger detected
		IF (SIf.Cur.dinNumOfHangersInBuffer <= 0)  AND (SIf.In.bolHangerDetected.intern) THEN
			SIf.Cur.dinNumOfHangersInBuffer := 1;
		END_IF
	END_IF
	
	// If buffer full detected, set number of hangers in buffer to max. capacity
	IF ((SIf.Cur.bolBufferFull = TRUE) AND (SIf.Cfg.bolHasBufferFullSensor = TRUE)) THEN	
		SIf.Cur.dinNumOfHangersInBuffer:= Sif.Cfg.dinMaxCapacity;
	END_IF
	
	// Limit Counter to max capacity
	IF (SIf.Cur.dinNumOfHangersInBuffer > SIf.Cfg.dinMaxCapacity) THEN
		SIf.Cur.dinNumOfHangersInBuffer:= SIf.Cfg.dinMaxCapacity;
	END_IF
	
	// Counter shows max. capacity, buffer full not detected (used for Bugzilla ID 55)
	IF ((SIf.Cur.dinNumOfHangersInBuffer >= SIf.Cfg.dinMaxCapacity) AND (SIf.In.bolBufferFull.intern =FALSE) AND
		(SIf.Cur.bolBufferFull = FALSE) AND (SIf.Cfg.bolHasBufferFullSensor = TRUE)) THEN	
		// Buffer is not full, decrement dinNumOfHangersInBuffer
		SIf.Cur.dinNumOfHangersInBuffer:= SIf.Cfg.dinMaxCapacity-1;
	END_IF
	
	
	// Limit Counter to min capacity
	IF SIf.Cur.dinNumOfHangersInBuffer < 0 THEN
		SIf.Cur.dinNumOfHangersInBuffer:= 0;
	END_IF
	
	// calculate max number of hangers could release per pulse
	IF (SIf.Cur.dinNumOfHangersInBuffer<=SIf.Cfg.uinNumOfHangersPerPulse) THEN
		dinNumOfHangersToRelease := SIf.Cur.dinNumOfHangersInBuffer;
	ELSE
		dinNumOfHangersToRelease := SIf.Cfg.uinNumOfHangersPerPulse;
	END_IF
END_IF


// ----------------------------------------------------------------------------------
// Always change actions in Base Library
// ----------------------------------------------------------------------------------
// overrule error always from base -> no EOFF State!! in EOFF go to OFF
IF (me.StateMachine.intStateNext = cSTA_EOFFBusy) THEN
	IF (me.StateMachine.intState=cSTA_OFF) THEN
		me.StateMachine.intStateNext := cSTA_OFF;
	ELSE // stay in OFF
		me.StateMachine.intStateNext := cSTA_OFFBusy;
	END_IF
END_IF

// Conditions Always
IF (((me.Alarm.eActivAlmClass=E_AlmClass.EOFF) OR (me.Alarm.eActivAlmClass=E_AlmClass.OFF) OR (me.intCmd=cCMD_OFF))
		 AND (me.StateMachine.intState<>cSTA_ERROR) AND (me.StateMachine.intState<>cSTA_ERRORQuit) AND
		(me.StateMachine.intState<>cSTA_OFF) AND (me.StateMachine.intState<>cSTA_OFFBusy)) THEN
	// alarm evt EOFF, OFF or cmd off
	me.StateMachine.intStateNext := cSTA_OFFBusy;
END_IF
END_METHOD

PROPERTY BufferFull : BOOL
GET
BufferFull:= SIf.Cur.bolBufferFull;
END_GET
END_PROPERTY

METHOD FB_init : BOOL
VAR_INPUT
	///if TRUE, the retain variables are initialized (warm start / cold start)
	bInitRetains: BOOL;
	///if TRUE, the instance afterwards gets moved into the copy code (online change)
	bInCopyCode: BOOL;
END_VAR
VAR
	ii: UINT;
END_VAR
//------------------------------------------------------------------------------------------------------------------------
// to manually change in new FUB implementation!!!
// define valid commands for this controller
FOR ii:= 0 TO (SIZEOF(CIf.Job.aCmdList)/SIZEOF(CIf.Job.aCmdList[0])-1) BY 1 DO
	IF (CIf.Job.aCmdList[ii].intCmd=cCMD_INITIALIZED) THEN
		// found first empty array element
		EXIT;
	END_IF
END_FOR

CIf.Job.aCmdList[ii].intCmd := cCMD_STOP;
CIf.Job.aCmdList[ii].strName := 'Stop'; 
CIf.Job.aCmdList[ii].bolAvailable := TRUE;
ii := ii +1;
CIf.Job.aCmdList[ii].intCmd := STB_CmdState.cCMD_RELEASE_ALL;
CIf.Job.aCmdList[ii].strName := 'Release All';
CIf.Job.aCmdList[ii].bolAvailable := TRUE;
ii := ii +1;
CIf.Job.aCmdList[ii].intCmd := STB_CmdState.cCMD_RELEASE;
CIf.Job.aCmdList[ii].strName := 'Release';
CIf.Job.aCmdList[ii].bolAvailable := TRUE;

// set name of class/typ
CIf.Info.strType := 'FB_STB'; 

// set alarm class
SIf.Alm[1].eAlmClass := E_AlmClass.STOP;
SIf.Alm[1].strText := 'Timeout buffer emptying';
SIf.Alm[2].eAlmClass := E_AlmClass.STOP;
SIf.Alm[2].strText := 'interlock retract - movement stopped';
SIf.Alm[3].eAlmClass := E_AlmClass.STOP;
SIf.Alm[3].strText := 'Cylinder position lost. Hangers slip through';

//*******************************************************************************
// initial values
//*******************************************************************************

// software configuration
CIf.SwCfg.bolExist := TRUE;
CIf.SwCfg.bolSimulation := FALSE;

// parameter
SIf.Par.udiIntervalBufferEmptying_ms := 2000;
SIf.Par.udiPulseLengthValve_ms := 500;
SIf.Par.udiSensorTime_ms := 3000;
SIf.Par.udiTimeoutBufferEmptying_ms := 120000; // 2 min
SIf.Par.usiBuffermode := 1;
SIf.Par.udiReleaseAllTime_ms := 4000;
Sif.par.udiDebounceTime_ms:= 20;

// configuration
SIf.Cfg.bolHasBufferFullSensor := FALSE;
SIf.Cfg.bolHasHangerDetection:= TRUE;
SIf.Cfg.bolHasDecrementSensor:= FALSE;
SIf.Cfg.bolDisableBufferDelete:= FALSE;
SIf.Cfg.dinMaxCapacity:= 20;
SIf.Cfg.dinMaxNumOfHangers_PosMonitoring := 2;
SIf.Cfg.uinNumOfHangersPerPulse:= 1;
SIF.Cfg.bolCylPosLostMonitoring:= FALSE;
SIF.Cfg.bolReleaseAllNonPulse:= FALSE;
END_METHOD

METHOD PROTECTED getCmdState : STRING
VAR_INPUT
	intCmdState: INT;
	bolState: BOOL;
END_VAR
getCmdState := SUPER^.getCmdState(intCmdState:=intCmdState,bolState:=bolState); // get global/base defined cmds/states
IF (getCmdState='') THEN // global not defined get local
	// get string cmd/state string information in runtime
	IF (bolState=FALSE) THEN
		// cmd's
		CASE intCmdState OF
			STB_CmdState.cCMD_RELEASE_ALL: 
				getCmdState := 'cCMD_RELEASE_ALL';
			STB_CmdState.cCMD_RELEASE: 
				getCmdState := 'cCMD_RELEASE';
		END_CASE;
	ELSE
	
	// states
		CASE intCmdState OF
			STB_CmdState.cSTA_RELEASE_ALLBusy: 
				getCmdState := 'cSTA_RELEASE_ALLBusy';
			STB_CmdState.cSTA_RELEASE_ALL: 
				getCmdState := 'cSTA_RELEASE_ALL';
			STB_CmdState.cSTA_RELEASEBusy: 
				getCmdState := 'cSTA_RELEASEBusy';
			STB_CmdState.cCMD_RELEASE: 
				getCmdState := 'cCMD_RELEASE';
		
			// SUB States
			cSTA_SUB_INITIALIZED:
				getCmdState := 'cSTA_SUB_INITIALIZED';
			cSTA_SUB_HANGER_PASSING:
				getCmdState := 'cSTA_SUB_HANGER_PASSING';
			cSTA_SUB_HANGER_PASSED:
				getCmdState := 'cSTA_SUB_HANGER_PASSED';
											
		END_CASE;
	END_IF
END_IF
END_METHOD

METHOD getCtrlSIf : POINTER TO T_Ctrl_SIf_STB
getCtrlSIf := ADR(SIf);
END_METHOD

METHOD PROTECTED IoInBridge : BOOL
// digitale and analoge inputs read from hardware or forcing

SIf.In.bolHangerDetected.map := THIS^.In_bolHangerDetected;
SIf.In.bolBufferFull.map := THIS^.In_bolBufferFull;
SIf.In.bolDecrementCounter.map := THIS^.In_bolDecrementCounter;

IF (CIf.SwCfg.bolSimulation = FALSE) THEN
	getInBolDebounced(CIf.Job.bolIoForce, me.FUBInfo.udiSample_ms, Sif.par.udiDebounceTime_ms, ADR(SIf.In.bolHangerDetected));
	getInBolDebounced(CIf.Job.bolIoForce, me.FUBInfo.udiSample_ms, Sif.par.udiDebounceTime_ms, ADR(SIf.In.bolBufferFull));
	getInBolDebounced(CIf.Job.bolIoForce, me.FUBInfo.udiSample_ms, Sif.par.udiDebounceTime_ms, ADR(SIf.In.bolDecrementCounter));
	//ctrl.In.bol_PosSwitchBasicDefTyp.intern := getInBol(ctrl.ifc.Job.bol_Force ,ADR(ctrl.In.bol_PosSwitchBasicDefTyp);
ELSE
	//simulation of global IO
END_IF
END_METHOD

METHOD PROTECTED IoOutBridge : BOOL
// digitale and analoge inputs read from hardware or forcing
IF (CIf.SwCfg.bolSimulation = FALSE) THEN
	setOutBol(CIf.Job.bolIoForce ,ADR(SIf.Out.bolRetract));
	
	// check interlocks to prevent damages
	IF (CIf.Job.bolIlkOverwrite=FALSE) THEN
		IF (SIf.Ilk.bolRetract=TRUE) THEN
			// switch off?
			IF (SIf.Out.bolRetract.map = TRUE) THEN
				// Set alarm: SIf.Alm[2].strText := 'interlock retract - movement stopped';				
				pfbAlarmCtrl^.setAlarm(CIf.Info.intCtrlId,2,0,ADR(SIf.Alm),E_AlmState.RST,CIf.Job.eMe_ActivAlmClass);				
			END_IF
			SIf.Out.bolRetract.map := FALSE;
		END_IF	
	END_IF
	THIS^.Out_bolRetract := SIf.Out.bolRetract.map;
	


	setOutBol(CIf.Job.bolIoForce ,ADR(SIf.Out.bolRetract2));
	
	// check interlocks to prevent damages
	IF (CIf.Job.bolIlkOverwrite=FALSE) THEN
		IF (SIf.Ilk.bolRetract=TRUE) THEN
			// switch off?
			IF (SIf.Out.bolRetract2.map = TRUE) THEN
				// Set alarm: SIf.Alm[2].strText := 'interlock retract - movement stopped';				
				pfbAlarmCtrl^.setAlarm(CIf.Info.intCtrlId,2,0,ADR(SIf.Alm),E_AlmState.RST,CIf.Job.eMe_ActivAlmClass);				
			END_IF
			SIf.Out.bolRetract2.map := FALSE;
		END_IF	
	END_IF
	THIS^.Out_bolRetract2 := SIf.Out.bolRetract2.map;
	
END_IF
END_METHOD

PROPERTY MaxCapacity : DINT
GET
MaxCapacity:= SIf.Cfg.dinMaxCapacity;
END_GET
END_PROPERTY

PROPERTY NumOfHangers : DINT
GET
NumOfHangers:= SIf.Cur.dinNumOfHangersInBuffer;
END_GET
END_PROPERTY

METHOD PROTECTED sta_ERROR : BOOL
// state implemetation
//--------------------------------------------------------------------------------------
// Entry action
	IF (me.StateMachine.intState<>me.StateMachine.intStateLastCycle) THEN
		me.StateMachine.intStateHistory := me.StateMachine.intStateLastCycle; // -> possibillity to go back to state before error
		me.StateMachine.intStateLastCycle := me.StateMachine.intState;
		
	END_IF

//--------------------------------------------------------------------------------------
// Cyclic action
	IF (me.StateMachine.intState=me.StateMachine.intStateLastCycle) THEN
		
		// Switch valve off, cylinder back to extend position -> stop hanger
		SIf.Out.bolRetract.intern := FALSE;
		SIf.Out.bolRetract2.intern := TRUE;	
		
		// State Change Condition
		IF (CIf.Job.bolAlmReset = TRUE) THEN
			me.StateMachine.intStateNext := cSTA_ERRORQuit;
		END_IF
	END_IF

//--------------------------------------------------------------------------------------
// Exit action
	IF (me.StateMachine.intState<>me.StateMachine.intStateNext) THEN
		;
	END_IF
END_METHOD

METHOD PROTECTED sta_OFF : BOOL
// state implemetation
//--------------------------------------------------------------------------------------
// Entry action
	IF (me.StateMachine.intState<>me.StateMachine.intStateLastCycle) THEN
		me.StateMachine.intStateLastCycle := me.StateMachine.intState;
		
		// Reset total counter
		SIf.Cur.dinHangersPassedTotal:= 0;
	END_IF


//--------------------------------------------------------------------------------------
// Cyclic action
	IF (me.StateMachine.intState=me.StateMachine.intStateLastCycle) THEN
		
	
		// State Change Condition
		IF (me.Alarm.eActivAlmClass<>E_AlmClass.EOFF) AND (me.Alarm.eActivAlmClass<>E_AlmClass.OFF) THEN
			IF (me.intCmd=cCMD_STOP) THEN
				me.StateMachine.intStateNext :=  cSTA_STOPBusy;
			ELSIF (me.intCmd=STB_CmdState.cCMD_RELEASE) THEN 
				me.StateMachine.intStateNext := STB_CmdState.cSTA_RELEASEBusy;
			ELSIF(me.intCmd=STB_CmdState.cCMD_RELEASE_ALL) THEN
				me.StateMachine.intStateNext := STB_CmdState.cSTA_RELEASE_ALLBusy;
			END_IF
		END_IF
	END_IF


//--------------------------------------------------------------------------------------
// Exit action
	IF (me.StateMachine.intState<>me.StateMachine.intStateNext) THEN
		;
	END_IF
END_METHOD

METHOD PROTECTED sta_OFFBusy : BOOL
// state implemetation
//--------------------------------------------------------------------------------------
// Entry action
	IF (me.StateMachine.intState<>me.StateMachine.intStateLastCycle) THEN
		me.StateMachine.intStateLastCycle := me.StateMachine.intState;
			
	END_IF

//--------------------------------------------------------------------------------------
// Cyclic action
	IF (me.StateMachine.intState=me.StateMachine.intStateLastCycle) THEN
		
		// Switch valve off, cylinder back to extend position -> stop hanger
		SIf.Out.bolRetract.intern := FALSE;
		SIf.Out.bolRetract2.intern := TRUE;	
			
		// State Change Condition
		IF (FALSE) THEN
			;
		ELSIF (TRUE) THEN
			me.StateMachine.intStateNext := cSTA_OFF;
		END_IF
	END_IF


//--------------------------------------------------------------------------------------
// Exit action
	IF (me.StateMachine.intState<>me.StateMachine.intStateNext) THEN
		;
	END_IF
END_METHOD

METHOD PROTECTED sta_RELEASE : BOOL
// state implemetation
//--------------------------------------------------------------------------------------
// Entry action
	IF (me.StateMachine.intState<>me.StateMachine.intStateLastCycle) THEN
		me.StateMachine.intStateLastCycle := me.StateMachine.intState;
			
		;
	END_IF

//--------------------------------------------------------------------------------------
// Cyclic action
	IF (me.StateMachine.intState=me.StateMachine.intStateLastCycle) THEN
		
		// Switch valve off, cylinder back to extend position -> stop hanger
		SIf.Out.bolRetract.intern := FALSE;
		SIf.Out.bolRetract2.intern := TRUE;	
		
		// State Change Condition
		IF (me.intCmd=cCMD_STOP) THEN
			me.StateMachine.intStateNext := cSTA_STOPBusy;
		ELSIF(me.intCmd=STB_CmdState.cCMD_RELEASE_ALL) THEN
			me.StateMachine.intStateNext := STB_CmdState.cSTA_RELEASE_ALLBusy;
		END_IF
		
	END_IF

//--------------------------------------------------------------------------------------
// Exit action
	IF (me.StateMachine.intState<>me.StateMachine.intStateNext) THEN
		;
	END_IF
END_METHOD

METHOD PROTECTED sta_RELEASE_ALL : BOOL
// state implemetation
//--------------------------------------------------------------------------------------
// Entry action
	IF (me.StateMachine.intState<>me.StateMachine.intStateLastCycle) THEN
		me.StateMachine.intStateLastCycle := me.StateMachine.intState;	
		;
	END_IF

//--------------------------------------------------------------------------------------
// Cyclic action
	IF (me.StateMachine.intState=me.StateMachine.intStateLastCycle) THEN
		

		// State Change Condition
		IF ((me.intCmd=cCMD_STOP) OR (me.intCmd=STB_CmdState.cCMD_RELEASE)) THEN
			me.StateMachine.intStateNext := cSTA_STOPBusy;
		END_IF
	END_IF

//--------------------------------------------------------------------------------------
// Exit action
	IF (me.StateMachine.intState<>me.StateMachine.intStateNext) THEN
		;
	END_IF
END_METHOD

METHOD PROTECTED sta_RELEASE_ALLBusy : BOOL
// state implemetation
//--------------------------------------------------------------------------------------
// Entry action
	IF (me.StateMachine.intState<>me.StateMachine.intStateLastCycle) THEN
		me.StateMachine.intStateLastCycle := me.StateMachine.intState;
				
		dinNumOfHangersToRelease:= 0;
		dinSetNumOfHangersToRelease:= 0;
		
		// Reset package counter
		SIf.Cur.dinHangersPassedPackage:= 0;
	
		// Initialize sub state machine
		me.SubStateMachine.intState:= cSTA_SUB_INITIALIZED; 
		me.SubStateMachine.intStateNext:= cSTA_SUB_INITIALIZED;
	
	END_IF

//--------------------------------------------------------------------------------------
// Cyclic action
	IF (me.StateMachine.intState=me.StateMachine.intStateLastCycle) THEN
			
		//--------------------------------------------------------------------------------------
		// sub state machine for release all sequence
		CASE me.SubStateMachine.intState OF
			//--------------------------------------------------------------------------------------
			cSTA_SUB_INITIALIZED:
				// Entry action
				IF (me.SubStateMachine.intState<>me.SubStateMachine.intStateLastCycle) THEN
					me.SubStateMachine.intStateLastCycle := me.SubStateMachine.intState;							
					
